   STATUS[84].EXT.Operation := FALSE;
   STATUS[84].EXT.Forced := TRUE;
   STATUS[84].EXT.BIT29 := FALSE;
   STATUS[84].EXT.BIT30 := FALSE;
   STATUS[84].EXT.BIT31 := FALSE;
   STATUS[84].EXT.ModeBit1 := FALSE;
   STATUS[84].EXT.ModeBit2 := FALSE;
   STATUS[84].EXT.ModeBit3 := FALSE;
   STATUS[84].EXT.BIT19 := FALSE;
   STATUS[84].EXT.BIT20 := FALSE;
   STATUS[84].EXT.AlarmSuppressed := FALSE;
   STATUS[84].EXT.AlarmPresent := FALSE;
   STATUS[84].EXT.AlarmFailUnAck := TRUE;
   STATUS[84].Status := 190;
   STATUS[84].TimeStamp := 16#1AEC;
   STATUS[85].EXT.AlarmWarnUnAck := FALSE;
   STATUS[85].EXT.AckRequired := FALSE;
   STATUS[85].EXT.Maintanence := FALSE;
   STATUS[85].EXT.Operation := TRUE;
   STATUS[85].EXT.Forced := FALSE;
   STATUS[85].EXT.BIT29 := FALSE;
   STATUS[85].EXT.BIT30 := FALSE;
   STATUS[85].EXT.BIT31 := FALSE;
   STATUS[85].EXT.ModeBit1 := FALSE;
   STATUS[85].EXT.ModeBit2 := FALSE;
   STATUS[85].EXT.ModeBit3 := FALSE;
   STATUS[85].EXT.BIT19 := FALSE;
   STATUS[85].EXT.BIT20 := FALSE;
   STATUS[85].EXT.AlarmSuppressed := FALSE;
   STATUS[85].EXT.AlarmPresent := FALSE;
   STATUS[85].EXT.AlarmFailUnAck := FALSE;
   STATUS[85].Status := 1;
   STATUS[85].TimeStamp := 16#3928;
   STATUS[86].EXT.AlarmWarnUnAck := FALSE;
   STATUS[86].EXT.AckRequired := FALSE;
   STATUS[86].EXT.Maintanence := FALSE;
   STATUS[86].EXT.Operation := TRUE;
   STATUS[86].EXT.Forced := FALSE;
   STATUS[86].EXT.BIT29 := FALSE;
   STATUS[86].EXT.BIT30 := FALSE;
   STATUS[86].EXT.BIT31 := FALSE;
   STATUS[86].EXT.ModeBit1 := FALSE;
   STATUS[86].EXT.ModeBit2 := FALSE;
   STATUS[86].EXT.ModeBit3 := FALSE;
   STATUS[86].EXT.BIT19 := FALSE;
   STATUS[86].EXT.BIT20 := FALSE;
   STATUS[86].EXT.AlarmSuppressed := FALSE;
   STATUS[86].EXT.AlarmPresent := FALSE;
   STATUS[86].EXT.AlarmFailUnAck := FALSE;
   STATUS[86].Status := 1;
   STATUS[86].TimeStamp := 16#3928;
   STATUS[87].EXT.AlarmWarnUnAck := FALSE;
   STATUS[87].EXT.AckRequired := FALSE;
   STATUS[87].EXT.Maintanence := FALSE;
   STATUS[87].EXT.Operation := FALSE;
   STATUS[87].EXT.Forced := FALSE;
   STATUS[87].EXT.BIT29 := FALSE;
   STATUS[87].EXT.BIT30 := FALSE;
   STATUS[87].EXT.BIT31 := FALSE;
   STATUS[87].EXT.ModeBit1 := FALSE;
   STATUS[87].EXT.ModeBit2 := FALSE;
   STATUS[87].EXT.ModeBit3 := FALSE;
   STATUS[87].EXT.BIT19 := FALSE;
   STATUS[87].EXT.BIT20 := FALSE;
   STATUS[87].EXT.AlarmSuppressed := TRUE;
   STATUS[87].EXT.AlarmPresent := FALSE;
   STATUS[87].EXT.AlarmFailUnAck := FALSE;
   STATUS[87].Status := 1;
   STATUS[87].TimeStamp := 16#84C0;
   STATUS[88].EXT.AlarmWarnUnAck := FALSE;
   STATUS[88].EXT.AckRequired := FALSE;
   STATUS[88].EXT.Maintanence := FALSE;
   STATUS[88].EXT.Operation := FALSE;
   STATUS[88].EXT.Forced := FALSE;
   STATUS[88].EXT.BIT29 := FALSE;
   STATUS[88].EXT.BIT30 := FALSE;
   STATUS[88].EXT.BIT31 := FALSE;
   STATUS[88].EXT.ModeBit1 := FALSE;
   STATUS[88].EXT.ModeBit2 := FALSE;
   STATUS[88].EXT.ModeBit3 := FALSE;
   STATUS[88].EXT.BIT19 := FALSE;
   STATUS[88].EXT.BIT20 := FALSE;
   STATUS[88].EXT.AlarmSuppressed := TRUE;
   STATUS[88].EXT.AlarmPresent := FALSE;
   STATUS[88].EXT.AlarmFailUnAck := FALSE;
   STATUS[88].Status := 1;
   STATUS[88].TimeStamp := 16#84BF;
   STATUS[89].EXT.AlarmWarnUnAck := FALSE;
   STATUS[89].EXT.AckRequired := FALSE;
   STATUS[89].EXT.Maintanence := FALSE;
   STATUS[89].EXT.Operation := FALSE;
   STATUS[89].EXT.Forced := TRUE;
   STATUS[89].EXT.BIT29 := FALSE;
   STATUS[89].EXT.BIT30 := FALSE;
   STATUS[89].EXT.BIT31 := FALSE;
   STATUS[89].EXT.ModeBit1 := FALSE;
   STATUS[89].EXT.ModeBit2 := FALSE;
   STATUS[89].EXT.ModeBit3 := FALSE;
   STATUS[89].EXT.BIT19 := FALSE;
   STATUS[89].EXT.BIT20 := FALSE;
   STATUS[89].EXT.AlarmSuppressed := FALSE;
   STATUS[89].EXT.AlarmPresent := FALSE;
   STATUS[89].EXT.AlarmFailUnAck := TRUE;
   STATUS[89].Status := 190;
   STATUS[89].TimeStamp := 16#71E9;
   STATUS[90].EXT.AlarmWarnUnAck := FALSE;
   STATUS[90].EXT.AckRequired := FALSE;
   STATUS[90].EXT.Maintanence := FALSE;
   STATUS[90].EXT.Operation := FALSE;
   STATUS[90].EXT.Forced := TRUE;
   STATUS[90].EXT.BIT29 := FALSE;
   STATUS[90].EXT.BIT30 := FALSE;
   STATUS[90].EXT.BIT31 := FALSE;
   STATUS[90].EXT.ModeBit1 := FALSE;
   STATUS[90].EXT.ModeBit2 := FALSE;
   STATUS[90].EXT.ModeBit3 := FALSE;
   STATUS[90].EXT.BIT19 := FALSE;
   STATUS[90].EXT.BIT20 := FALSE;
   STATUS[90].EXT.AlarmSuppressed := FALSE;
   STATUS[90].EXT.AlarmPresent := FALSE;
   STATUS[90].EXT.AlarmFailUnAck := TRUE;
   STATUS[90].Status := 190;
   STATUS[90].TimeStamp := 16#7C0C;
   STATUS[91].EXT.AlarmWarnUnAck := FALSE;
   STATUS[91].EXT.AckRequired := FALSE;
   STATUS[91].EXT.Maintanence := FALSE;
   STATUS[91].EXT.Operation := FALSE;
   STATUS[91].EXT.Forced := TRUE;
   STATUS[91].EXT.BIT29 := FALSE;
   STATUS[91].EXT.BIT30 := FALSE;
   STATUS[91].EXT.BIT31 := FALSE;
   STATUS[91].EXT.ModeBit1 := FALSE;
   STATUS[91].EXT.ModeBit2 := FALSE;
   STATUS[91].EXT.ModeBit3 := FALSE;
   STATUS[91].EXT.BIT19 := FALSE;
   STATUS[91].EXT.BIT20 := FALSE;
   STATUS[91].EXT.AlarmSuppressed := FALSE;
   STATUS[91].EXT.AlarmPresent := FALSE;
   STATUS[91].EXT.AlarmFailUnAck := TRUE;
   STATUS[91].Status := 190;
   STATUS[91].TimeStamp := 16#7882;
   STATUS[92].EXT.AlarmWarnUnAck := FALSE;
   STATUS[92].EXT.AckRequired := FALSE;
   STATUS[92].EXT.Maintanence := FALSE;
   STATUS[92].EXT.Operation := FALSE;
   STATUS[92].EXT.Forced := TRUE;
   STATUS[92].EXT.BIT29 := FALSE;
   STATUS[92].EXT.BIT30 := FALSE;
   STATUS[92].EXT.BIT31 := FALSE;
   STATUS[92].EXT.ModeBit1 := FALSE;
   STATUS[92].EXT.ModeBit2 := FALSE;
   STATUS[92].EXT.ModeBit3 := FALSE;
   STATUS[92].EXT.BIT19 := FALSE;
   STATUS[92].EXT.BIT20 := FALSE;
   STATUS[92].EXT.AlarmSuppressed := FALSE;
   STATUS[92].EXT.AlarmPresent := FALSE;
   STATUS[92].EXT.AlarmFailUnAck := TRUE;
   STATUS[92].Status := 190;
   STATUS[92].TimeStamp := 16#7534;
   STATUS[93].EXT.AlarmWarnUnAck := FALSE;
   STATUS[93].EXT.AckRequired := FALSE;
   STATUS[93].EXT.Maintanence := FALSE;
   STATUS[93].EXT.Operation := FALSE;
   STATUS[93].EXT.Forced := TRUE;
   STATUS[93].EXT.BIT29 := FALSE;
   STATUS[93].EXT.BIT30 := FALSE;
   STATUS[93].EXT.BIT31 := FALSE;
   STATUS[93].EXT.ModeBit1 := FALSE;
   STATUS[93].EXT.ModeBit2 := FALSE;
   STATUS[93].EXT.ModeBit3 := FALSE;
   STATUS[93].EXT.BIT19 := FALSE;
   STATUS[93].EXT.BIT20 := FALSE;
   STATUS[93].EXT.AlarmSuppressed := FALSE;
   STATUS[93].EXT.AlarmPresent := FALSE;
   STATUS[93].EXT.AlarmFailUnAck := TRUE;
   STATUS[93].Status := 190;
   STATUS[93].TimeStamp := 16#8187;
   STATUS[94].EXT.AlarmWarnUnAck := FALSE;
   STATUS[94].EXT.AckRequired := TRUE;
   STATUS[94].EXT.Maintanence := FALSE;
   STATUS[94].EXT.Operation := FALSE;
   STATUS[94].EXT.Forced := FALSE;
   STATUS[94].EXT.BIT29 := FALSE;
   STATUS[94].EXT.BIT30 := FALSE;
   STATUS[94].EXT.BIT31 := FALSE;
   STATUS[94].EXT.ModeBit1 := FALSE;
   STATUS[94].EXT.ModeBit2 := FALSE;
   STATUS[94].EXT.ModeBit3 := FALSE;
   STATUS[94].EXT.BIT19 := FALSE;
   STATUS[94].EXT.BIT20 := FALSE;
   STATUS[94].EXT.AlarmSuppressed := FALSE;
   STATUS[94].EXT.AlarmPresent := FALSE;
   STATUS[94].EXT.AlarmFailUnAck := TRUE;
   STATUS[94].Status := 231;
   STATUS[94].TimeStamp := 16#8854;
   STATUS[95].EXT.AlarmWarnUnAck := FALSE;
   STATUS[95].EXT.AckRequired := FALSE;
   STATUS[95].EXT.Maintanence := FALSE;
   STATUS[95].EXT.Operation := FALSE;
   STATUS[95].EXT.Forced := TRUE;
   STATUS[95].EXT.BIT29 := FALSE;
   STATUS[95].EXT.BIT30 := FALSE;
   STATUS[95].EXT.BIT31 := FALSE;
   STATUS[95].EXT.ModeBit1 := FALSE;
   STATUS[95].EXT.ModeBit2 := FALSE;
   STATUS[95].EXT.ModeBit3 := FALSE;
   STATUS[95].EXT.BIT19 := FALSE;
   STATUS[95].EXT.BIT20 := FALSE;
   STATUS[95].EXT.AlarmSuppressed := FALSE;
   STATUS[95].EXT.AlarmPresent := FALSE;
   STATUS[95].EXT.AlarmFailUnAck := TRUE;
   STATUS[95].Status := 190;
   STATUS[95].TimeStamp := 16#611D;
   STATUS[96].EXT.AlarmWarnUnAck := FALSE;
   STATUS[96].EXT.AckRequired := FALSE;
   STATUS[96].EXT.Maintanence := FALSE;
   STATUS[96].EXT.Operation := FALSE;
   STATUS[96].EXT.Forced := TRUE;
   STATUS[96].EXT.BIT29 := FALSE;
   STATUS[96].EXT.BIT30 := FALSE;
   STATUS[96].EXT.BIT31 := FALSE;
   STATUS[96].EXT.ModeBit1 := FALSE;
   STATUS[96].EXT.ModeBit2 := FALSE;
   STATUS[96].EXT.ModeBit3 := FALSE;
   STATUS[96].EXT.BIT19 := FALSE;
   STATUS[96].EXT.BIT20 := FALSE;
   STATUS[96].EXT.AlarmSuppressed := FALSE;
   STATUS[96].EXT.AlarmPresent := FALSE;
   STATUS[96].EXT.AlarmFailUnAck := TRUE;
   STATUS[96].Status := 190;
   STATUS[96].TimeStamp := 16#692D;
   STATUS[97].EXT.AlarmWarnUnAck := FALSE;
   STATUS[97].EXT.AckRequired := FALSE;
   STATUS[97].EXT.Maintanence := FALSE;
   STATUS[97].EXT.Operation := FALSE;
   STATUS[97].EXT.Forced := TRUE;
   STATUS[97].EXT.BIT29 := FALSE;
   STATUS[97].EXT.BIT30 := FALSE;
   STATUS[97].EXT.BIT31 := FALSE;
   STATUS[97].EXT.ModeBit1 := FALSE;
   STATUS[97].EXT.ModeBit2 := FALSE;
   STATUS[97].EXT.ModeBit3 := FALSE;
   STATUS[97].EXT.BIT19 := FALSE;
   STATUS[97].EXT.BIT20 := FALSE;
   STATUS[97].EXT.AlarmSuppressed := FALSE;
   STATUS[97].EXT.AlarmPresent := FALSE;
   STATUS[97].EXT.AlarmFailUnAck := TRUE;
   STATUS[97].Status := 190;
   STATUS[97].TimeStamp := 16#661E;
   STATUS[98].EXT.AlarmWarnUnAck := FALSE;
   STATUS[98].EXT.AckRequired := FALSE;
   STATUS[98].EXT.Maintanence := FALSE;
   STATUS[98].EXT.Operation := FALSE;
   STATUS[98].EXT.Forced := TRUE;
   STATUS[98].EXT.BIT29 := FALSE;
   STATUS[98].EXT.BIT30 := FALSE;
   STATUS[98].EXT.BIT31 := FALSE;
   STATUS[98].EXT.ModeBit1 := FALSE;
   STATUS[98].EXT.ModeBit2 := FALSE;
   STATUS[98].EXT.ModeBit3 := FALSE;
   STATUS[98].EXT.BIT19 := FALSE;
   STATUS[98].EXT.BIT20 := FALSE;
   STATUS[98].EXT.AlarmSuppressed := FALSE;
   STATUS[98].EXT.AlarmPresent := FALSE;
   STATUS[98].EXT.AlarmFailUnAck := TRUE;
   STATUS[98].Status := 190;
   STATUS[98].TimeStamp := 16#6F16;
   STATUS[99].EXT.AlarmWarnUnAck := FALSE;
   STATUS[99].EXT.AckRequired := FALSE;
   STATUS[99].EXT.Maintanence := FALSE;
   STATUS[99].EXT.Operation := FALSE;
   STATUS[99].EXT.Forced := TRUE;
   STATUS[99].EXT.BIT29 := FALSE;
   STATUS[99].EXT.BIT30 := FALSE;
   STATUS[99].EXT.BIT31 := FALSE;
   STATUS[99].EXT.ModeBit1 := FALSE;
   STATUS[99].EXT.ModeBit2 := FALSE;
   STATUS[99].EXT.ModeBit3 := FALSE;
   STATUS[99].EXT.BIT19 := FALSE;
   STATUS[99].EXT.BIT20 := FALSE;
   STATUS[99].EXT.AlarmSuppressed := FALSE;
   STATUS[99].EXT.AlarmPresent := FALSE;
   STATUS[99].EXT.AlarmFailUnAck := TRUE;
   STATUS[99].Status := 190;
   STATUS[99].TimeStamp := 16#4FA7;
   STATUS[100].EXT.AlarmWarnUnAck := FALSE;
   STATUS[100].EXT.AckRequired := FALSE;
   STATUS[100].EXT.Maintanence := FALSE;
   STATUS[100].EXT.Operation := FALSE;
   STATUS[100].EXT.Forced := TRUE;
   STATUS[100].EXT.BIT29 := FALSE;
   STATUS[100].EXT.BIT30 := FALSE;
   STATUS[100].EXT.BIT31 := FALSE;
   STATUS[100].EXT.ModeBit1 := FALSE;
   STATUS[100].EXT.ModeBit2 := FALSE;
   STATUS[100].EXT.ModeBit3 := FALSE;
   STATUS[100].EXT.BIT19 := FALSE;
   STATUS[100].EXT.BIT20 := FALSE;
   STATUS[100].EXT.AlarmSuppressed := FALSE;
   STATUS[100].EXT.AlarmPresent := FALSE;
   STATUS[100].EXT.AlarmFailUnAck := TRUE;
   STATUS[100].Status := 190;
   STATUS[100].TimeStamp := 16#8403;
   STATUS[101].EXT.AlarmWarnUnAck := FALSE;
   STATUS[101].EXT.AckRequired := FALSE;
   STATUS[101].EXT.Maintanence := FALSE;
   STATUS[101].EXT.Operation := FALSE;
   STATUS[101].EXT.Forced := TRUE;
   STATUS[101].EXT.BIT29 := FALSE;
   STATUS[101].EXT.BIT30 := FALSE;
   STATUS[101].EXT.BIT31 := FALSE;
   STATUS[101].EXT.ModeBit1 := FALSE;
   STATUS[101].EXT.ModeBit2 := FALSE;
   STATUS[101].EXT.ModeBit3 := FALSE;
   STATUS[101].EXT.BIT19 := FALSE;
   STATUS[101].EXT.BIT20 := FALSE;
   STATUS[101].EXT.AlarmSuppressed := FALSE;
   STATUS[101].EXT.AlarmPresent := FALSE;
   STATUS[101].EXT.AlarmFailUnAck := TRUE;
   STATUS[101].Status := 190;
   STATUS[101].TimeStamp := 16#6C19;
   STATUS[102].EXT.AlarmWarnUnAck := FALSE;
   STATUS[102].EXT.AckRequired := FALSE;
   STATUS[102].EXT.Maintanence := FALSE;
   STATUS[102].EXT.Operation := FALSE;
   STATUS[102].EXT.Forced := TRUE;
   STATUS[102].EXT.BIT29 := FALSE;
   STATUS[102].EXT.BIT30 := FALSE;
   STATUS[102].EXT.BIT31 := FALSE;
   STATUS[102].EXT.ModeBit1 := FALSE;
   STATUS[102].EXT.ModeBit2 := FALSE;
   STATUS[102].EXT.ModeBit3 := FALSE;
   STATUS[102].EXT.BIT19 := FALSE;
   STATUS[102].EXT.BIT20 := FALSE;
   STATUS[102].EXT.AlarmSuppressed := FALSE;
   STATUS[102].EXT.AlarmPresent := FALSE;
   STATUS[102].EXT.AlarmFailUnAck := TRUE;
   STATUS[102].Status := 190;
   STATUS[102].TimeStamp := 16#7EB8;
   STATUS[103].EXT.AlarmWarnUnAck := FALSE;
   STATUS[103].EXT.AckRequired := FALSE;
   STATUS[103].EXT.Maintanence := FALSE;
   STATUS[103].EXT.Operation := TRUE;
   STATUS[103].EXT.Forced := FALSE;
   STATUS[103].EXT.BIT29 := FALSE;
   STATUS[103].EXT.BIT30 := FALSE;
   STATUS[103].EXT.BIT31 := FALSE;
   STATUS[103].EXT.ModeBit1 := FALSE;
   STATUS[103].EXT.ModeBit2 := FALSE;
   STATUS[103].EXT.ModeBit3 := FALSE;
   STATUS[103].EXT.BIT19 := FALSE;
   STATUS[103].EXT.BIT20 := FALSE;
   STATUS[103].EXT.AlarmSuppressed := FALSE;
   STATUS[103].EXT.AlarmPresent := FALSE;
   STATUS[103].EXT.AlarmFailUnAck := FALSE;
   STATUS[103].Status := 1;
   STATUS[103].TimeStamp := 16#3928;
   STATUS[104].EXT.AlarmWarnUnAck := FALSE;
   STATUS[104].EXT.AckRequired := FALSE;
   STATUS[104].EXT.Maintanence := FALSE;
   STATUS[104].EXT.Operation := TRUE;
   STATUS[104].EXT.Forced := FALSE;
   STATUS[104].EXT.BIT29 := FALSE;
   STATUS[104].EXT.BIT30 := FALSE;
   STATUS[104].EXT.BIT31 := FALSE;
   STATUS[104].EXT.ModeBit1 := FALSE;
   STATUS[104].EXT.ModeBit2 := FALSE;
   STATUS[104].EXT.ModeBit3 := FALSE;
   STATUS[104].EXT.BIT19 := FALSE;
   STATUS[104].EXT.BIT20 := FALSE;
   STATUS[104].EXT.AlarmSuppressed := FALSE;
   STATUS[104].EXT.AlarmPresent := FALSE;
   STATUS[104].EXT.AlarmFailUnAck := FALSE;
   STATUS[104].Status := 1;
   STATUS[104].TimeStamp := 16#3928;
   STATUS[105].EXT.AlarmWarnUnAck := FALSE;
   STATUS[105].EXT.AckRequired := FALSE;
   STATUS[105].EXT.Maintanence := FALSE;
   STATUS[105].EXT.Operation := TRUE;
   STATUS[105].EXT.Forced := FALSE;
   STATUS[105].EXT.BIT29 := FALSE;
   STATUS[105].EXT.BIT30 := FALSE;
   STATUS[105].EXT.BIT31 := FALSE;
   STATUS[105].EXT.ModeBit1 := FALSE;
   STATUS[105].EXT.ModeBit2 := FALSE;
   STATUS[105].EXT.ModeBit3 := FALSE;
   STATUS[105].EXT.BIT19 := FALSE;
   STATUS[105].EXT.BIT20 := FALSE;
   STATUS[105].EXT.AlarmSuppressed := FALSE;
   STATUS[105].EXT.AlarmPresent := FALSE;
   STATUS[105].EXT.AlarmFailUnAck := FALSE;
   STATUS[105].Status := 1;
   STATUS[105].TimeStamp := 16#3928;
   STATUS[106].EXT.AlarmWarnUnAck := FALSE;
   STATUS[106].EXT.AckRequired := FALSE;
   STATUS[106].EXT.Maintanence := FALSE;
   STATUS[106].EXT.Operation := TRUE;
   STATUS[106].EXT.Forced := FALSE;
   STATUS[106].EXT.BIT29 := FALSE;
   STATUS[106].EXT.BIT30 := FALSE;
   STATUS[106].EXT.BIT31 := FALSE;
   STATUS[106].EXT.ModeBit1 := FALSE;
   STATUS[106].EXT.ModeBit2 := FALSE;
   STATUS[106].EXT.ModeBit3 := FALSE;
   STATUS[106].EXT.BIT19 := FALSE;
   STATUS[106].EXT.BIT20 := FALSE;
   STATUS[106].EXT.AlarmSuppressed := FALSE;
   STATUS[106].EXT.AlarmPresent := FALSE;
   STATUS[106].EXT.AlarmFailUnAck := FALSE;
   STATUS[106].Status := 1;
   STATUS[106].TimeStamp := 16#3928;
   STATUS[107].EXT.AlarmWarnUnAck := FALSE;
   STATUS[107].EXT.AckRequired := FALSE;
   STATUS[107].EXT.Maintanence := FALSE;
   STATUS[107].EXT.Operation := TRUE;
   STATUS[107].EXT.Forced := FALSE;
   STATUS[107].EXT.BIT29 := FALSE;
   STATUS[107].EXT.BIT30 := FALSE;
   STATUS[107].EXT.BIT31 := FALSE;
   STATUS[107].EXT.ModeBit1 := FALSE;
   STATUS[107].EXT.ModeBit2 := FALSE;
   STATUS[107].EXT.ModeBit3 := FALSE;
   STATUS[107].EXT.BIT19 := FALSE;
   STATUS[107].EXT.BIT20 := FALSE;
   STATUS[107].EXT.AlarmSuppressed := FALSE;
   STATUS[107].EXT.AlarmPresent := FALSE;
   STATUS[107].EXT.AlarmFailUnAck := FALSE;
   STATUS[107].Status := 1;
   STATUS[107].TimeStamp := 16#3928;
   STATUS[108].EXT.AlarmWarnUnAck := FALSE;
   STATUS[108].EXT.AckRequired := FALSE;
   STATUS[108].EXT.Maintanence := FALSE;
   STATUS[108].EXT.Operation := FALSE;
   STATUS[108].EXT.Forced := FALSE;
   STATUS[108].EXT.BIT29 := FALSE;
   STATUS[108].EXT.BIT30 := FALSE;
   STATUS[108].EXT.BIT31 := FALSE;
   STATUS[108].EXT.ModeBit1 := FALSE;
   STATUS[108].EXT.ModeBit2 := FALSE;
   STATUS[108].EXT.ModeBit3 := FALSE;
   STATUS[108].EXT.BIT19 := FALSE;
   STATUS[108].EXT.BIT20 := FALSE;
   STATUS[108].EXT.AlarmSuppressed := TRUE;
   STATUS[108].EXT.AlarmPresent := TRUE;
   STATUS[108].EXT.AlarmFailUnAck := TRUE;
   STATUS[108].Status := 201;
   STATUS[108].TimeStamp := 16#CE77;
   STATUS[109].EXT.AlarmWarnUnAck := FALSE;
   STATUS[109].EXT.AckRequired := FALSE;
   STATUS[109].EXT.Maintanence := FALSE;
   STATUS[109].EXT.Operation := FALSE;
   STATUS[109].EXT.Forced := TRUE;
   STATUS[109].EXT.BIT29 := FALSE;
   STATUS[109].EXT.BIT30 := FALSE;
   STATUS[109].EXT.BIT31 := FALSE;
   STATUS[109].EXT.ModeBit1 := FALSE;
   STATUS[109].EXT.ModeBit2 := FALSE;
   STATUS[109].EXT.ModeBit3 := FALSE;
   STATUS[109].EXT.BIT19 := FALSE;
   STATUS[109].EXT.BIT20 := FALSE;
   STATUS[109].EXT.AlarmSuppressed := FALSE;
   STATUS[109].EXT.AlarmPresent := FALSE;
   STATUS[109].EXT.AlarmFailUnAck := TRUE;
   STATUS[109].Status := 190;
   STATUS[109].TimeStamp := 16#D712;
   STATUS[110].EXT.AlarmWarnUnAck := FALSE;
   STATUS[110].EXT.AckRequired := FALSE;
   STATUS[110].EXT.Maintanence := FALSE;
   STATUS[110].EXT.Operation := FALSE;
   STATUS[110].EXT.Forced := TRUE;
   STATUS[110].EXT.BIT29 := FALSE;
   STATUS[110].EXT.BIT30 := FALSE;
   STATUS[110].EXT.BIT31 := FALSE;
   STATUS[110].EXT.ModeBit1 := FALSE;
   STATUS[110].EXT.ModeBit2 := FALSE;
   STATUS[110].EXT.ModeBit3 := FALSE;
   STATUS[110].EXT.BIT19 := FALSE;
   STATUS[110].EXT.BIT20 := FALSE;
   STATUS[110].EXT.AlarmSuppressed := FALSE;
   STATUS[110].EXT.AlarmPresent := FALSE;
   STATUS[110].EXT.AlarmFailUnAck := TRUE;
   STATUS[110].Status := 190;
   STATUS[110].TimeStamp := 16#969A;
   STATUS[111].EXT.AlarmWarnUnAck := FALSE;
   STATUS[111].EXT.AckRequired := FALSE;
   STATUS[111].EXT.Maintanence := FALSE;
   STATUS[111].EXT.Operation := FALSE;
   STATUS[111].EXT.Forced := FALSE;
   STATUS[111].EXT.BIT29 := FALSE;
   STATUS[111].EXT.BIT30 := FALSE;
   STATUS[111].EXT.BIT31 := FALSE;
   STATUS[111].EXT.ModeBit1 := FALSE;
   STATUS[111].EXT.ModeBit2 := FALSE;
   STATUS[111].EXT.ModeBit3 := FALSE;
   STATUS[111].EXT.BIT19 := FALSE;
   STATUS[111].EXT.BIT20 := FALSE;
   STATUS[111].EXT.AlarmSuppressed := TRUE;
   STATUS[111].EXT.AlarmPresent := FALSE;
   STATUS[111].EXT.AlarmFailUnAck := FALSE;
   STATUS[111].Status := 1;
   STATUS[111].TimeStamp := 16#9BB5;
   STATUS[112].EXT.AlarmWarnUnAck := FALSE;
   STATUS[112].EXT.AckRequired := FALSE;
   STATUS[112].EXT.Maintanence := FALSE;
   STATUS[112].EXT.Operation := FALSE;
   STATUS[112].EXT.Forced := TRUE;
   STATUS[112].EXT.BIT29 := FALSE;
   STATUS[112].EXT.BIT30 := FALSE;
   STATUS[112].EXT.BIT31 := FALSE;
   STATUS[112].EXT.ModeBit1 := FALSE;
   STATUS[112].EXT.ModeBit2 := FALSE;
   STATUS[112].EXT.ModeBit3 := FALSE;
   STATUS[112].EXT.BIT19 := FALSE;
   STATUS[112].EXT.BIT20 := FALSE;
   STATUS[112].EXT.AlarmSuppressed := FALSE;
   STATUS[112].EXT.AlarmPresent := FALSE;
   STATUS[112].EXT.AlarmFailUnAck := TRUE;
   STATUS[112].Status := 190;
   STATUS[112].TimeStamp := 16#87AE;
   STATUS[113].EXT.AlarmWarnUnAck := FALSE;
   STATUS[113].EXT.AckRequired := FALSE;
   STATUS[113].EXT.Maintanence := FALSE;
   STATUS[113].EXT.Operation := FALSE;
   STATUS[113].EXT.Forced := FALSE;
   STATUS[113].EXT.BIT29 := FALSE;
   STATUS[113].EXT.BIT30 := FALSE;
   STATUS[113].EXT.BIT31 := FALSE;
   STATUS[113].EXT.ModeBit1 := FALSE;
   STATUS[113].EXT.ModeBit2 := FALSE;
   STATUS[113].EXT.ModeBit3 := FALSE;
   STATUS[113].EXT.BIT19 := FALSE;
   STATUS[113].EXT.BIT20 := FALSE;
   STATUS[113].EXT.AlarmSuppressed := FALSE;
   STATUS[113].EXT.AlarmPresent := FALSE;
   STATUS[113].EXT.AlarmFailUnAck := FALSE;
   STATUS[113].Status := -22466;
   STATUS[113].TimeStamp := 16#84BA;
   STATUS[114].EXT.AlarmWarnUnAck := FALSE;
   STATUS[114].EXT.AckRequired := FALSE;
   STATUS[114].EXT.Maintanence := FALSE;
   STATUS[114].EXT.Operation := TRUE;
   STATUS[114].EXT.Forced := FALSE;
   STATUS[114].EXT.BIT29 := FALSE;
   STATUS[114].EXT.BIT30 := FALSE;
   STATUS[114].EXT.BIT31 := FALSE;
   STATUS[114].EXT.ModeBit1 := FALSE;
   STATUS[114].EXT.ModeBit2 := FALSE;
   STATUS[114].EXT.ModeBit3 := FALSE;
   STATUS[114].EXT.BIT19 := FALSE;
   STATUS[114].EXT.BIT20 := FALSE;
   STATUS[114].EXT.AlarmSuppressed := FALSE;
   STATUS[114].EXT.AlarmPresent := FALSE;
   STATUS[114].EXT.AlarmFailUnAck := FALSE;
   STATUS[114].Status := 4177;
   STATUS[114].TimeStamp := 16#583C;
   STATUS[115].EXT.AlarmWarnUnAck := FALSE;
   STATUS[115].EXT.AckRequired := FALSE;
   STATUS[115].EXT.Maintanence := FALSE;
   STATUS[115].EXT.Operation := TRUE;
   STATUS[115].EXT.Forced := FALSE;
   STATUS[115].EXT.BIT29 := FALSE;
   STATUS[115].EXT.BIT30 := FALSE;
   STATUS[115].EXT.BIT31 := FALSE;
   STATUS[115].EXT.ModeBit1 := FALSE;
   STATUS[115].EXT.ModeBit2 := FALSE;
   STATUS[115].EXT.ModeBit3 := FALSE;
   STATUS[115].EXT.BIT19 := FALSE;
   STATUS[115].EXT.BIT20 := FALSE;
   STATUS[115].EXT.AlarmSuppressed := FALSE;
   STATUS[115].EXT.AlarmPresent := FALSE;
   STATUS[115].EXT.AlarmFailUnAck := FALSE;
   STATUS[115].Status := 4177;
   STATUS[115].TimeStamp := 16#5ACA;
   STATUS[116].EXT.AlarmWarnUnAck := FALSE;
   STATUS[116].EXT.AckRequired := FALSE;
   STATUS[116].EXT.Maintanence := FALSE;
   STATUS[116].EXT.Operation := FALSE;
   STATUS[116].EXT.Forced := FALSE;
   STATUS[116].EXT.BIT29 := FALSE;
   STATUS[116].EXT.BIT30 := FALSE;
   STATUS[116].EXT.BIT31 := FALSE;
   STATUS[116].EXT.ModeBit1 := FALSE;
   STATUS[116].EXT.ModeBit2 := FALSE;
   STATUS[116].EXT.ModeBit3 := FALSE;
   STATUS[116].EXT.BIT19 := FALSE;
   STATUS[116].EXT.BIT20 := FALSE;
   STATUS[116].EXT.AlarmSuppressed := TRUE;
   STATUS[116].EXT.AlarmPresent := FALSE;
   STATUS[116].EXT.AlarmFailUnAck := FALSE;
   STATUS[116].Status := 1;
   STATUS[116].TimeStamp := 16#84BF;
   STATUS[117].EXT.AlarmWarnUnAck := FALSE;
   STATUS[117].EXT.AckRequired := FALSE;
   STATUS[117].EXT.Maintanence := FALSE;
   STATUS[117].EXT.Operation := FALSE;
   STATUS[117].EXT.Forced := FALSE;
   STATUS[117].EXT.BIT29 := FALSE;
   STATUS[117].EXT.BIT30 := FALSE;
   STATUS[117].EXT.BIT31 := FALSE;
   STATUS[117].EXT.ModeBit1 := FALSE;
   STATUS[117].EXT.ModeBit2 := FALSE;
   STATUS[117].EXT.ModeBit3 := FALSE;
   STATUS[117].EXT.BIT19 := FALSE;
   STATUS[117].EXT.BIT20 := FALSE;
   STATUS[117].EXT.AlarmSuppressed := TRUE;
   STATUS[117].EXT.AlarmPresent := TRUE;
   STATUS[117].EXT.AlarmFailUnAck := TRUE;
   STATUS[117].Status := 201;
   STATUS[117].TimeStamp := 16#E23A;
   STATUS[118].EXT.AlarmWarnUnAck := FALSE;
   STATUS[118].EXT.AckRequired := FALSE;
   STATUS[118].EXT.Maintanence := FALSE;
   STATUS[118].EXT.Operation := FALSE;
   STATUS[118].EXT.Forced := FALSE;
   STATUS[118].EXT.BIT29 := FALSE;
   STATUS[118].EXT.BIT30 := FALSE;
   STATUS[118].EXT.BIT31 := FALSE;
   STATUS[118].EXT.ModeBit1 := FALSE;
   STATUS[118].EXT.ModeBit2 := FALSE;
   STATUS[118].EXT.ModeBit3 := FALSE;
   STATUS[118].EXT.BIT19 := FALSE;
   STATUS[118].EXT.BIT20 := FALSE;
   STATUS[118].EXT.AlarmSuppressed := TRUE;
   STATUS[118].EXT.AlarmPresent := TRUE;
   STATUS[118].EXT.AlarmFailUnAck := TRUE;
   STATUS[118].Status := 212;
   STATUS[118].TimeStamp := 16#3928;
   STATUS[119].EXT.AlarmWarnUnAck := FALSE;
   STATUS[119].EXT.AckRequired := FALSE;
   STATUS[119].EXT.Maintanence := FALSE;
   STATUS[119].EXT.Operation := FALSE;
   STATUS[119].EXT.Forced := FALSE;
   STATUS[119].EXT.BIT29 := FALSE;
   STATUS[119].EXT.BIT30 := FALSE;
   STATUS[119].EXT.BIT31 := FALSE;
   STATUS[119].EXT.ModeBit1 := FALSE;
   STATUS[119].EXT.ModeBit2 := FALSE;
   STATUS[119].EXT.ModeBit3 := FALSE;
   STATUS[119].EXT.BIT19 := FALSE;
   STATUS[119].EXT.BIT20 := FALSE;
   STATUS[119].EXT.AlarmSuppressed := TRUE;
   STATUS[119].EXT.AlarmPresent := TRUE;
   STATUS[119].EXT.AlarmFailUnAck := TRUE;
   STATUS[119].Status := 212;
   STATUS[119].TimeStamp := 16#3928;
   STATUS[120].EXT.AlarmWarnUnAck := FALSE;
   STATUS[120].EXT.AckRequired := FALSE;
   STATUS[120].EXT.Maintanence := FALSE;
   STATUS[120].EXT.Operation := FALSE;
   STATUS[120].EXT.Forced := FALSE;
   STATUS[120].EXT.BIT29 := FALSE;
   STATUS[120].EXT.BIT30 := FALSE;
   STATUS[120].EXT.BIT31 := FALSE;
   STATUS[120].EXT.ModeBit1 := FALSE;
   STATUS[120].EXT.ModeBit2 := FALSE;
   STATUS[120].EXT.ModeBit3 := FALSE;
   STATUS[120].EXT.BIT19 := FALSE;
   STATUS[120].EXT.BIT20 := FALSE;
   STATUS[120].EXT.AlarmSuppressed := TRUE;
   STATUS[120].EXT.AlarmPresent := TRUE;
   STATUS[120].EXT.AlarmFailUnAck := TRUE;
   STATUS[120].Status := 212;
   STATUS[120].TimeStamp := 16#3928;
   STATUS[121].EXT.AlarmWarnUnAck := FALSE;
   STATUS[121].EXT.AckRequired := FALSE;
   STATUS[121].EXT.Maintanence := FALSE;
   STATUS[121].EXT.Operation := FALSE;
   STATUS[121].EXT.Forced := FALSE;
   STATUS[121].EXT.BIT29 := FALSE;
   STATUS[121].EXT.BIT30 := FALSE;
   STATUS[121].EXT.BIT31 := FALSE;
   STATUS[121].EXT.ModeBit1 := FALSE;
   STATUS[121].EXT.ModeBit2 := FALSE;
   STATUS[121].EXT.ModeBit3 := FALSE;
   STATUS[121].EXT.BIT19 := FALSE;
   STATUS[121].EXT.BIT20 := FALSE;
   STATUS[121].EXT.AlarmSuppressed := TRUE;
   STATUS[121].EXT.AlarmPresent := TRUE;
   STATUS[121].EXT.AlarmFailUnAck := TRUE;
   STATUS[121].Status := 212;
   STATUS[121].TimeStamp := 16#3928;
   STATUS[122].EXT.AlarmWarnUnAck := FALSE;
   STATUS[122].EXT.AckRequired := FALSE;
   STATUS[122].EXT.Maintanence := FALSE;
   STATUS[122].EXT.Operation := FALSE;
   STATUS[122].EXT.Forced := FALSE;
   STATUS[122].EXT.BIT29 := FALSE;
   STATUS[122].EXT.BIT30 := FALSE;
   STATUS[122].EXT.BIT31 := FALSE;
   STATUS[122].EXT.ModeBit1 := FALSE;
   STATUS[122].EXT.ModeBit2 := FALSE;
   STATUS[122].EXT.ModeBit3 := FALSE;
   STATUS[122].EXT.BIT19 := FALSE;
   STATUS[122].EXT.BIT20 := FALSE;
   STATUS[122].EXT.AlarmSuppressed := TRUE;
   STATUS[122].EXT.AlarmPresent := TRUE;
   STATUS[122].EXT.AlarmFailUnAck := TRUE;
   STATUS[122].Status := 212;
   STATUS[122].TimeStamp := 16#3928;
   STATUS[123].EXT.AlarmWarnUnAck := FALSE;
   STATUS[123].EXT.AckRequired := FALSE;
   STATUS[123].EXT.Maintanence := FALSE;
   STATUS[123].EXT.Operation := FALSE;
   STATUS[123].EXT.Forced := FALSE;
   STATUS[123].EXT.BIT29 := FALSE;
   STATUS[123].EXT.BIT30 := FALSE;
   STATUS[123].EXT.BIT31 := FALSE;
   STATUS[123].EXT.ModeBit1 := FALSE;
   STATUS[123].EXT.ModeBit2 := FALSE;
   STATUS[123].EXT.ModeBit3 := FALSE;
   STATUS[123].EXT.BIT19 := FALSE;
   STATUS[123].EXT.BIT20 := FALSE;
   STATUS[123].EXT.AlarmSuppressed := TRUE;
   STATUS[123].EXT.AlarmPresent := TRUE;
   STATUS[123].EXT.AlarmFailUnAck := TRUE;
   STATUS[123].Status := 207;
   STATUS[123].TimeStamp := 16#84C0;
   STATUS[124].EXT.AlarmWarnUnAck := FALSE;
   STATUS[124].EXT.AckRequired := FALSE;
   STATUS[124].EXT.Maintanence := FALSE;
   STATUS[124].EXT.Operation := TRUE;
   STATUS[124].EXT.Forced := FALSE;
   STATUS[124].EXT.BIT29 := FALSE;
   STATUS[124].EXT.BIT30 := FALSE;
   STATUS[124].EXT.BIT31 := FALSE;
   STATUS[124].EXT.ModeBit1 := FALSE;
   STATUS[124].EXT.ModeBit2 := FALSE;
   STATUS[124].EXT.ModeBit3 := FALSE;
   STATUS[124].EXT.BIT19 := FALSE;
   STATUS[124].EXT.BIT20 := FALSE;
   STATUS[124].EXT.AlarmSuppressed := FALSE;
   STATUS[124].EXT.AlarmPresent := FALSE;
   STATUS[124].EXT.AlarmFailUnAck := FALSE;
   STATUS[124].Status := 1;
   STATUS[124].TimeStamp := 16#3928;
   STATUS[125].EXT.AlarmWarnUnAck := FALSE;
   STATUS[125].EXT.AckRequired := FALSE;
   STATUS[125].EXT.Maintanence := FALSE;
   STATUS[125].EXT.Operation := FALSE;
   STATUS[125].EXT.Forced := FALSE;
   STATUS[125].EXT.BIT29 := FALSE;
   STATUS[125].EXT.BIT30 := FALSE;
   STATUS[125].EXT.BIT31 := FALSE;
   STATUS[125].EXT.ModeBit1 := FALSE;
   STATUS[125].EXT.ModeBit2 := FALSE;
   STATUS[125].EXT.ModeBit3 := FALSE;
   STATUS[125].EXT.BIT19 := FALSE;
   STATUS[125].EXT.BIT20 := FALSE;
   STATUS[125].EXT.AlarmSuppressed := FALSE;
   STATUS[125].EXT.AlarmPresent := FALSE;
   STATUS[125].EXT.AlarmFailUnAck := FALSE;
   STATUS[125].Status := 0;
   STATUS[125].TimeStamp := 16#0000;
   STATUS[126].EXT.AlarmWarnUnAck := FALSE;
   STATUS[126].EXT.AckRequired := FALSE;
   STATUS[126].EXT.Maintanence := FALSE;
   STATUS[126].EXT.Operation := FALSE;
   STATUS[126].EXT.Forced := FALSE;
   STATUS[126].EXT.BIT29 := FALSE;
   STATUS[126].EXT.BIT30 := FALSE;
   STATUS[126].EXT.BIT31 := FALSE;
   STATUS[126].EXT.ModeBit1 := FALSE;
   STATUS[126].EXT.ModeBit2 := FALSE;
   STATUS[126].EXT.ModeBit3 := FALSE;
   STATUS[126].EXT.BIT19 := FALSE;
   STATUS[126].EXT.BIT20 := FALSE;
   STATUS[126].EXT.AlarmSuppressed := FALSE;
   STATUS[126].EXT.AlarmPresent := FALSE;
   STATUS[126].EXT.AlarmFailUnAck := FALSE;
   STATUS[126].Status := 0;
   STATUS[126].TimeStamp := 16#0000;
   STATUS[127].EXT.AlarmWarnUnAck := FALSE;
   STATUS[127].EXT.AckRequired := FALSE;
   STATUS[127].EXT.Maintanence := FALSE;
   STATUS[127].EXT.Operation := FALSE;
   STATUS[127].EXT.Forced := FALSE;
   STATUS[127].EXT.BIT29 := FALSE;
   STATUS[127].EXT.BIT30 := FALSE;
   STATUS[127].EXT.BIT31 := FALSE;
   STATUS[127].EXT.ModeBit1 := FALSE;
   STATUS[127].EXT.ModeBit2 := FALSE;
   STATUS[127].EXT.ModeBit3 := FALSE;
   STATUS[127].EXT.BIT19 := FALSE;
   STATUS[127].EXT.BIT20 := FALSE;
   STATUS[127].EXT.AlarmSuppressed := FALSE;
   STATUS[127].EXT.AlarmPresent := FALSE;
   STATUS[127].EXT.AlarmFailUnAck := FALSE;
   STATUS[127].Status := 0;
   STATUS[127].TimeStamp := 16#0000;
   STATUS[128].EXT.AlarmWarnUnAck := FALSE;
   STATUS[128].EXT.AckRequired := FALSE;
   STATUS[128].EXT.Maintanence := FALSE;
   STATUS[128].EXT.Operation := FALSE;
   STATUS[128].EXT.Forced := FALSE;
   STATUS[128].EXT.BIT29 := FALSE;
   STATUS[128].EXT.BIT30 := FALSE;
   STATUS[128].EXT.BIT31 := FALSE;
   STATUS[128].EXT.ModeBit1 := FALSE;
   STATUS[128].EXT.ModeBit2 := FALSE;
   STATUS[128].EXT.ModeBit3 := FALSE;
   STATUS[128].EXT.BIT19 := FALSE;
   STATUS[128].EXT.BIT20 := FALSE;
   STATUS[128].EXT.AlarmSuppressed := FALSE;
   STATUS[128].EXT.AlarmPresent := FALSE;
   STATUS[128].EXT.AlarmFailUnAck := FALSE;
   STATUS[128].Status := 0;
   STATUS[128].TimeStamp := 16#0000;
   STATUS[129].EXT.AlarmWarnUnAck := FALSE;
   STATUS[129].EXT.AckRequired := FALSE;
   STATUS[129].EXT.Maintanence := FALSE;
   STATUS[129].EXT.Operation := FALSE;
   STATUS[129].EXT.Forced := FALSE;
   STATUS[129].EXT.BIT29 := FALSE;
   STATUS[129].EXT.BIT30 := FALSE;
   STATUS[129].EXT.BIT31 := FALSE;
   STATUS[129].EXT.ModeBit1 := FALSE;
   STATUS[129].EXT.ModeBit2 := FALSE;
   STATUS[129].EXT.ModeBit3 := FALSE;
   STATUS[129].EXT.BIT19 := FALSE;
   STATUS[129].EXT.BIT20 := FALSE;
   STATUS[129].EXT.AlarmSuppressed := FALSE;
   STATUS[129].EXT.AlarmPresent := FALSE;
   STATUS[129].EXT.AlarmFailUnAck := FALSE;
   STATUS[129].Status := 0;
   STATUS[129].TimeStamp := 16#0000;
   STATUS[130].EXT.AlarmWarnUnAck := FALSE;
   STATUS[130].EXT.AckRequired := FALSE;
   STATUS[130].EXT.Maintanence := FALSE;
   STATUS[130].EXT.Operation := FALSE;
   STATUS[130].EXT.Forced := FALSE;
   STATUS[130].EXT.BIT29 := FALSE;
   STATUS[130].EXT.BIT30 := FALSE;
   STATUS[130].EXT.BIT31 := FALSE;
   STATUS[130].EXT.ModeBit1 := FALSE;
   STATUS[130].EXT.ModeBit2 := FALSE;
   STATUS[130].EXT.ModeBit3 := FALSE;
   STATUS[130].EXT.BIT19 := FALSE;
   STATUS[130].EXT.BIT20 := FALSE;
   STATUS[130].EXT.AlarmSuppressed := FALSE;
   STATUS[130].EXT.AlarmPresent := FALSE;
   STATUS[130].EXT.AlarmFailUnAck := FALSE;
   STATUS[130].Status := 0;
   STATUS[130].TimeStamp := 16#0000;
   STATUS[131].EXT.AlarmWarnUnAck := FALSE;
   STATUS[131].EXT.AckRequired := FALSE;
   STATUS[131].EXT.Maintanence := FALSE;
   STATUS[131].EXT.Operation := FALSE;
   STATUS[131].EXT.Forced := FALSE;
   STATUS[131].EXT.BIT29 := FALSE;
   STATUS[131].EXT.BIT30 := FALSE;
   STATUS[131].EXT.BIT31 := FALSE;
   STATUS[131].EXT.ModeBit1 := FALSE;
   STATUS[131].EXT.ModeBit2 := FALSE;
   STATUS[131].EXT.ModeBit3 := FALSE;
   STATUS[131].EXT.BIT19 := FALSE;
   STATUS[131].EXT.BIT20 := FALSE;
   STATUS[131].EXT.AlarmSuppressed := FALSE;
   STATUS[131].EXT.AlarmPresent := FALSE;
   STATUS[131].EXT.AlarmFailUnAck := FALSE;
   STATUS[131].Status := 0;
   STATUS[131].TimeStamp := 16#0000;
   STATUS[132].EXT.AlarmWarnUnAck := FALSE;
   STATUS[132].EXT.AckRequired := FALSE;
   STATUS[132].EXT.Maintanence := FALSE;
   STATUS[132].EXT.Operation := FALSE;
   STATUS[132].EXT.Forced := FALSE;
   STATUS[132].EXT.BIT29 := FALSE;
   STATUS[132].EXT.BIT30 := FALSE;
   STATUS[132].EXT.BIT31 := FALSE;
   STATUS[132].EXT.ModeBit1 := FALSE;
   STATUS[132].EXT.ModeBit2 := FALSE;
   STATUS[132].EXT.ModeBit3 := FALSE;
   STATUS[132].EXT.BIT19 := FALSE;
   STATUS[132].EXT.BIT20 := FALSE;
   STATUS[132].EXT.AlarmSuppressed := FALSE;
   STATUS[132].EXT.AlarmPresent := FALSE;
   STATUS[132].EXT.AlarmFailUnAck := FALSE;
   STATUS[132].Status := 0;
   STATUS[132].TimeStamp := 16#0000;
   STATUS[133].EXT.AlarmWarnUnAck := FALSE;
   STATUS[133].EXT.AckRequired := FALSE;
   STATUS[133].EXT.Maintanence := FALSE;
   STATUS[133].EXT.Operation := FALSE;
   STATUS[133].EXT.Forced := FALSE;
   STATUS[133].EXT.BIT29 := FALSE;
   STATUS[133].EXT.BIT30 := FALSE;
   STATUS[133].EXT.BIT31 := FALSE;
   STATUS[133].EXT.ModeBit1 := FALSE;
   STATUS[133].EXT.ModeBit2 := FALSE;
   STATUS[133].EXT.ModeBit3 := FALSE;
   STATUS[133].EXT.BIT19 := FALSE;
   STATUS[133].EXT.BIT20 := FALSE;
   STATUS[133].EXT.AlarmSuppressed := FALSE;
   STATUS[133].EXT.AlarmPresent := FALSE;
   STATUS[133].EXT.AlarmFailUnAck := FALSE;
   STATUS[133].Status := 0;
   STATUS[133].TimeStamp := 16#0000;
   STATUS[134].EXT.AlarmWarnUnAck := FALSE;
   STATUS[134].EXT.AckRequired := FALSE;
   STATUS[134].EXT.Maintanence := FALSE;
   STATUS[134].EXT.Operation := FALSE;
   STATUS[134].EXT.Forced := FALSE;
   STATUS[134].EXT.BIT29 := FALSE;
   STATUS[134].EXT.BIT30 := FALSE;
   STATUS[134].EXT.BIT31 := FALSE;
   STATUS[134].EXT.ModeBit1 := FALSE;
   STATUS[134].EXT.ModeBit2 := FALSE;
   STATUS[134].EXT.ModeBit3 := FALSE;
   STATUS[134].EXT.BIT19 := FALSE;
   STATUS[134].EXT.BIT20 := FALSE;
   STATUS[134].EXT.AlarmSuppressed := FALSE;
   STATUS[134].EXT.AlarmPresent := FALSE;
   STATUS[134].EXT.AlarmFailUnAck := FALSE;
   STATUS[134].Status := 0;
   STATUS[134].TimeStamp := 16#0000;
   STATUS[135].EXT.AlarmWarnUnAck := FALSE;
   STATUS[135].EXT.AckRequired := FALSE;
   STATUS[135].EXT.Maintanence := FALSE;
   STATUS[135].EXT.Operation := FALSE;
   STATUS[135].EXT.Forced := FALSE;
   STATUS[135].EXT.BIT29 := FALSE;
   STATUS[135].EXT.BIT30 := FALSE;
   STATUS[135].EXT.BIT31 := FALSE;
   STATUS[135].EXT.ModeBit1 := FALSE;
   STATUS[135].EXT.ModeBit2 := FALSE;
   STATUS[135].EXT.ModeBit3 := FALSE;
   STATUS[135].EXT.BIT19 := FALSE;
   STATUS[135].EXT.BIT20 := FALSE;
   STATUS[135].EXT.AlarmSuppressed := FALSE;
   STATUS[135].EXT.AlarmPresent := FALSE;
   STATUS[135].EXT.AlarmFailUnAck := FALSE;
   STATUS[135].Status := 0;
   STATUS[135].TimeStamp := 16#0000;
   STATUS[136].EXT.AlarmWarnUnAck := FALSE;
   STATUS[136].EXT.AckRequired := FALSE;
   STATUS[136].EXT.Maintanence := FALSE;
   STATUS[136].EXT.Operation := FALSE;
   STATUS[136].EXT.Forced := FALSE;
   STATUS[136].EXT.BIT29 := FALSE;
   STATUS[136].EXT.BIT30 := FALSE;
   STATUS[136].EXT.BIT31 := FALSE;
   STATUS[136].EXT.ModeBit1 := FALSE;
   STATUS[136].EXT.ModeBit2 := FALSE;
   STATUS[136].EXT.ModeBit3 := FALSE;
   STATUS[136].EXT.BIT19 := FALSE;
   STATUS[136].EXT.BIT20 := FALSE;
   STATUS[136].EXT.AlarmSuppressed := FALSE;
   STATUS[136].EXT.AlarmPresent := FALSE;
   STATUS[136].EXT.AlarmFailUnAck := FALSE;
   STATUS[136].Status := 0;
   STATUS[136].TimeStamp := 16#0000;
   STATUS[137].EXT.AlarmWarnUnAck := FALSE;
   STATUS[137].EXT.AckRequired := FALSE;
   STATUS[137].EXT.Maintanence := FALSE;
   STATUS[137].EXT.Operation := FALSE;
   STATUS[137].EXT.Forced := FALSE;
   STATUS[137].EXT.BIT29 := FALSE;
   STATUS[137].EXT.BIT30 := FALSE;
   STATUS[137].EXT.BIT31 := FALSE;
   STATUS[137].EXT.ModeBit1 := FALSE;
   STATUS[137].EXT.ModeBit2 := FALSE;
   STATUS[137].EXT.ModeBit3 := FALSE;
   STATUS[137].EXT.BIT19 := FALSE;
   STATUS[137].EXT.BIT20 := FALSE;
   STATUS[137].EXT.AlarmSuppressed := FALSE;
   STATUS[137].EXT.AlarmPresent := FALSE;
   STATUS[137].EXT.AlarmFailUnAck := FALSE;
   STATUS[137].Status := 0;
   STATUS[137].TimeStamp := 16#0000;
   STATUS[138].EXT.AlarmWarnUnAck := FALSE;
   STATUS[138].EXT.AckRequired := FALSE;
   STATUS[138].EXT.Maintanence := FALSE;
   STATUS[138].EXT.Operation := FALSE;
   STATUS[138].EXT.Forced := FALSE;
   STATUS[138].EXT.BIT29 := FALSE;
   STATUS[138].EXT.BIT30 := FALSE;
   STATUS[138].EXT.BIT31 := FALSE;
   STATUS[138].EXT.ModeBit1 := FALSE;
   STATUS[138].EXT.ModeBit2 := FALSE;
   STATUS[138].EXT.ModeBit3 := FALSE;
   STATUS[138].EXT.BIT19 := FALSE;
   STATUS[138].EXT.BIT20 := FALSE;
   STATUS[138].EXT.AlarmSuppressed := FALSE;
   STATUS[138].EXT.AlarmPresent := FALSE;
   STATUS[138].EXT.AlarmFailUnAck := FALSE;
   STATUS[138].Status := 0;
   STATUS[138].TimeStamp := 16#0000;
   STATUS[139].EXT.AlarmWarnUnAck := FALSE;
   STATUS[139].EXT.AckRequired := FALSE;
   STATUS[139].EXT.Maintanence := FALSE;
   STATUS[139].EXT.Operation := FALSE;
   STATUS[139].EXT.Forced := FALSE;
   STATUS[139].EXT.BIT29 := FALSE;
   STATUS[139].EXT.BIT30 := FALSE;
   STATUS[139].EXT.BIT31 := FALSE;
   STATUS[139].EXT.ModeBit1 := FALSE;
   STATUS[139].EXT.ModeBit2 := FALSE;
   STATUS[139].EXT.ModeBit3 := FALSE;
   STATUS[139].EXT.BIT19 := FALSE;
   STATUS[139].EXT.BIT20 := FALSE;
   STATUS[139].EXT.AlarmSuppressed := FALSE;
   STATUS[139].EXT.AlarmPresent := FALSE;
   STATUS[139].EXT.AlarmFailUnAck := FALSE;
   STATUS[139].Status := 0;
   STATUS[139].TimeStamp := 16#0000;
   STATUS[140].EXT.AlarmWarnUnAck := FALSE;
   STATUS[140].EXT.AckRequired := FALSE;
   STATUS[140].EXT.Maintanence := FALSE;
   STATUS[140].EXT.Operation := FALSE;
   STATUS[140].EXT.Forced := FALSE;
   STATUS[140].EXT.BIT29 := FALSE;
   STATUS[140].EXT.BIT30 := FALSE;
   STATUS[140].EXT.BIT31 := FALSE;
   STATUS[140].EXT.ModeBit1 := FALSE;
   STATUS[140].EXT.ModeBit2 := FALSE;
   STATUS[140].EXT.ModeBit3 := FALSE;
   STATUS[140].EXT.BIT19 := FALSE;
   STATUS[140].EXT.BIT20 := FALSE;
   STATUS[140].EXT.AlarmSuppressed := FALSE;
   STATUS[140].EXT.AlarmPresent := FALSE;
   STATUS[140].EXT.AlarmFailUnAck := FALSE;
   STATUS[140].Status := 0;
   STATUS[140].TimeStamp := 16#0000;
   STATUS[141].EXT.AlarmWarnUnAck := FALSE;
   STATUS[141].EXT.AckRequired := FALSE;
   STATUS[141].EXT.Maintanence := FALSE;
   STATUS[141].EXT.Operation := FALSE;
   STATUS[141].EXT.Forced := FALSE;
   STATUS[141].EXT.BIT29 := FALSE;
   STATUS[141].EXT.BIT30 := FALSE;
   STATUS[141].EXT.BIT31 := FALSE;
   STATUS[141].EXT.ModeBit1 := FALSE;
   STATUS[141].EXT.ModeBit2 := FALSE;
   STATUS[141].EXT.ModeBit3 := FALSE;
   STATUS[141].EXT.BIT19 := FALSE;
   STATUS[141].EXT.BIT20 := FALSE;
   STATUS[141].EXT.AlarmSuppressed := FALSE;
   STATUS[141].EXT.AlarmPresent := FALSE;
   STATUS[141].EXT.AlarmFailUnAck := FALSE;
   STATUS[141].Status := 0;
   STATUS[141].TimeStamp := 16#0000;
   STATUS[142].EXT.AlarmWarnUnAck := FALSE;
   STATUS[142].EXT.AckRequired := FALSE;
   STATUS[142].EXT.Maintanence := FALSE;
   STATUS[142].EXT.Operation := FALSE;
   STATUS[142].EXT.Forced := FALSE;
   STATUS[142].EXT.BIT29 := FALSE;
   STATUS[142].EXT.BIT30 := FALSE;
   STATUS[142].EXT.BIT31 := FALSE;
   STATUS[142].EXT.ModeBit1 := FALSE;
   STATUS[142].EXT.ModeBit2 := FALSE;
   STATUS[142].EXT.ModeBit3 := FALSE;
   STATUS[142].EXT.BIT19 := FALSE;
   STATUS[142].EXT.BIT20 := FALSE;
   STATUS[142].EXT.AlarmSuppressed := FALSE;
   STATUS[142].EXT.AlarmPresent := FALSE;
   STATUS[142].EXT.AlarmFailUnAck := FALSE;
   STATUS[142].Status := 0;
   STATUS[142].TimeStamp := 16#0000;
   STATUS[143].EXT.AlarmWarnUnAck := FALSE;
   STATUS[143].EXT.AckRequired := FALSE;
   STATUS[143].EXT.Maintanence := FALSE;
   STATUS[143].EXT.Operation := FALSE;
   STATUS[143].EXT.Forced := FALSE;
   STATUS[143].EXT.BIT29 := FALSE;
   STATUS[143].EXT.BIT30 := FALSE;
   STATUS[143].EXT.BIT31 := FALSE;
   STATUS[143].EXT.ModeBit1 := FALSE;
   STATUS[143].EXT.ModeBit2 := FALSE;
   STATUS[143].EXT.ModeBit3 := FALSE;
   STATUS[143].EXT.BIT19 := FALSE;
   STATUS[143].EXT.BIT20 := FALSE;
   STATUS[143].EXT.AlarmSuppressed := FALSE;
   STATUS[143].EXT.AlarmPresent := FALSE;
   STATUS[143].EXT.AlarmFailUnAck := FALSE;
   STATUS[143].Status := 0;
   STATUS[143].TimeStamp := 16#0000;
   STATUS[144].EXT.AlarmWarnUnAck := FALSE;
   STATUS[144].EXT.AckRequired := FALSE;
   STATUS[144].EXT.Maintanence := FALSE;
   STATUS[144].EXT.Operation := FALSE;
   STATUS[144].EXT.Forced := FALSE;
   STATUS[144].EXT.BIT29 := FALSE;
   STATUS[144].EXT.BIT30 := FALSE;
   STATUS[144].EXT.BIT31 := FALSE;
   STATUS[144].EXT.ModeBit1 := FALSE;
   STATUS[144].EXT.ModeBit2 := FALSE;
   STATUS[144].EXT.ModeBit3 := FALSE;
   STATUS[144].EXT.BIT19 := FALSE;
   STATUS[144].EXT.BIT20 := FALSE;
   STATUS[144].EXT.AlarmSuppressed := FALSE;
   STATUS[144].EXT.AlarmPresent := FALSE;
   STATUS[144].EXT.AlarmFailUnAck := FALSE;
   STATUS[144].Status := 0;
   STATUS[144].TimeStamp := 16#0000;
   STATUS[145].EXT.AlarmWarnUnAck := FALSE;
   STATUS[145].EXT.AckRequired := FALSE;
   STATUS[145].EXT.Maintanence := FALSE;
   STATUS[145].EXT.Operation := FALSE;
   STATUS[145].EXT.Forced := FALSE;
   STATUS[145].EXT.BIT29 := FALSE;
   STATUS[145].EXT.BIT30 := FALSE;
   STATUS[145].EXT.BIT31 := FALSE;
   STATUS[145].EXT.ModeBit1 := FALSE;
   STATUS[145].EXT.ModeBit2 := FALSE;
   STATUS[145].EXT.ModeBit3 := FALSE;
   STATUS[145].EXT.BIT19 := FALSE;
   STATUS[145].EXT.BIT20 := FALSE;
   STATUS[145].EXT.AlarmSuppressed := FALSE;
   STATUS[145].EXT.AlarmPresent := FALSE;
   STATUS[145].EXT.AlarmFailUnAck := FALSE;
   STATUS[145].Status := 0;
   STATUS[145].TimeStamp := 16#0000;
   STATUS[146].EXT.AlarmWarnUnAck := FALSE;
   STATUS[146].EXT.AckRequired := FALSE;
   STATUS[146].EXT.Maintanence := FALSE;
   STATUS[146].EXT.Operation := FALSE;
   STATUS[146].EXT.Forced := FALSE;
   STATUS[146].EXT.BIT29 := FALSE;
   STATUS[146].EXT.BIT30 := FALSE;
   STATUS[146].EXT.BIT31 := FALSE;
   STATUS[146].EXT.ModeBit1 := FALSE;
   STATUS[146].EXT.ModeBit2 := FALSE;
   STATUS[146].EXT.ModeBit3 := FALSE;
   STATUS[146].EXT.BIT19 := FALSE;
   STATUS[146].EXT.BIT20 := FALSE;
   STATUS[146].EXT.AlarmSuppressed := FALSE;
   STATUS[146].EXT.AlarmPresent := FALSE;
   STATUS[146].EXT.AlarmFailUnAck := FALSE;
   STATUS[146].Status := 0;
   STATUS[146].TimeStamp := 16#0000;
   STATUS[147].EXT.AlarmWarnUnAck := FALSE;
   STATUS[147].EXT.AckRequired := FALSE;
   STATUS[147].EXT.Maintanence := FALSE;
   STATUS[147].EXT.Operation := FALSE;
   STATUS[147].EXT.Forced := FALSE;
   STATUS[147].EXT.BIT29 := FALSE;
   STATUS[147].EXT.BIT30 := FALSE;
   STATUS[147].EXT.BIT31 := FALSE;
   STATUS[147].EXT.ModeBit1 := FALSE;
   STATUS[147].EXT.ModeBit2 := FALSE;
   STATUS[147].EXT.ModeBit3 := FALSE;
   STATUS[147].EXT.BIT19 := FALSE;
   STATUS[147].EXT.BIT20 := FALSE;
   STATUS[147].EXT.AlarmSuppressed := FALSE;
   STATUS[147].EXT.AlarmPresent := FALSE;
   STATUS[147].EXT.AlarmFailUnAck := FALSE;
   STATUS[147].Status := 0;
   STATUS[147].TimeStamp := 16#0000;
   STATUS[148].EXT.AlarmWarnUnAck := FALSE;
   STATUS[148].EXT.AckRequired := FALSE;
   STATUS[148].EXT.Maintanence := FALSE;
   STATUS[148].EXT.Operation := FALSE;
   STATUS[148].EXT.Forced := FALSE;
   STATUS[148].EXT.BIT29 := FALSE;
   STATUS[148].EXT.BIT30 := FALSE;
   STATUS[148].EXT.BIT31 := FALSE;
   STATUS[148].EXT.ModeBit1 := FALSE;
   STATUS[148].EXT.ModeBit2 := FALSE;
   STATUS[148].EXT.ModeBit3 := FALSE;
   STATUS[148].EXT.BIT19 := FALSE;
   STATUS[148].EXT.BIT20 := FALSE;
   STATUS[148].EXT.AlarmSuppressed := FALSE;
   STATUS[148].EXT.AlarmPresent := FALSE;
   STATUS[148].EXT.AlarmFailUnAck := FALSE;
   STATUS[148].Status := 0;
   STATUS[148].TimeStamp := 16#0000;
   STATUS[149].EXT.AlarmWarnUnAck := FALSE;
   STATUS[149].EXT.AckRequired := FALSE;
   STATUS[149].EXT.Maintanence := FALSE;
   STATUS[149].EXT.Operation := FALSE;
   STATUS[149].EXT.Forced := FALSE;
   STATUS[149].EXT.BIT29 := FALSE;
   STATUS[149].EXT.BIT30 := FALSE;
   STATUS[149].EXT.BIT31 := FALSE;
   STATUS[149].EXT.ModeBit1 := FALSE;
   STATUS[149].EXT.ModeBit2 := FALSE;
   STATUS[149].EXT.ModeBit3 := FALSE;
   STATUS[149].EXT.BIT19 := FALSE;
   STATUS[149].EXT.BIT20 := FALSE;
   STATUS[149].EXT.AlarmSuppressed := FALSE;
   STATUS[149].EXT.AlarmPresent := FALSE;
   STATUS[149].EXT.AlarmFailUnAck := FALSE;
   STATUS[149].Status := 0;
   STATUS[149].TimeStamp := 16#0000;
   STATUS[150].EXT.AlarmWarnUnAck := FALSE;
   STATUS[150].EXT.AckRequired := FALSE;
   STATUS[150].EXT.Maintanence := FALSE;
   STATUS[150].EXT.Operation := FALSE;
   STATUS[150].EXT.Forced := FALSE;
   STATUS[150].EXT.BIT29 := FALSE;
   STATUS[150].EXT.BIT30 := FALSE;
   STATUS[150].EXT.BIT31 := FALSE;
   STATUS[150].EXT.ModeBit1 := FALSE;
   STATUS[150].EXT.ModeBit2 := FALSE;
   STATUS[150].EXT.ModeBit3 := FALSE;
   STATUS[150].EXT.BIT19 := FALSE;
   STATUS[150].EXT.BIT20 := FALSE;
   STATUS[150].EXT.AlarmSuppressed := FALSE;
   STATUS[150].EXT.AlarmPresent := FALSE;
   STATUS[150].EXT.AlarmFailUnAck := FALSE;
   STATUS[150].Status := 0;
   STATUS[150].TimeStamp := 16#0000;
   STATUS[151].EXT.AlarmWarnUnAck := FALSE;
   STATUS[151].EXT.AckRequired := FALSE;
   STATUS[151].EXT.Maintanence := FALSE;
   STATUS[151].EXT.Operation := FALSE;
   STATUS[151].EXT.Forced := FALSE;
   STATUS[151].EXT.BIT29 := FALSE;
   STATUS[151].EXT.BIT30 := FALSE;
   STATUS[151].EXT.BIT31 := FALSE;
   STATUS[151].EXT.ModeBit1 := FALSE;
   STATUS[151].EXT.ModeBit2 := FALSE;
   STATUS[151].EXT.ModeBit3 := FALSE;
   STATUS[151].EXT.BIT19 := FALSE;
   STATUS[151].EXT.BIT20 := FALSE;
   STATUS[151].EXT.AlarmSuppressed := FALSE;
   STATUS[151].EXT.AlarmPresent := FALSE;
   STATUS[151].EXT.AlarmFailUnAck := FALSE;
   STATUS[151].Status := 0;
   STATUS[151].TimeStamp := 16#0000;
   STATUS[152].EXT.AlarmWarnUnAck := FALSE;
   STATUS[152].EXT.AckRequired := FALSE;
   STATUS[152].EXT.Maintanence := FALSE;
   STATUS[152].EXT.Operation := FALSE;
   STATUS[152].EXT.Forced := FALSE;
   STATUS[152].EXT.BIT29 := FALSE;
   STATUS[152].EXT.BIT30 := FALSE;
   STATUS[152].EXT.BIT31 := FALSE;
   STATUS[152].EXT.ModeBit1 := FALSE;
   STATUS[152].EXT.ModeBit2 := FALSE;
   STATUS[152].EXT.ModeBit3 := FALSE;
   STATUS[152].EXT.BIT19 := FALSE;
   STATUS[152].EXT.BIT20 := FALSE;
   STATUS[152].EXT.AlarmSuppressed := FALSE;
   STATUS[152].EXT.AlarmPresent := FALSE;
   STATUS[152].EXT.AlarmFailUnAck := FALSE;
   STATUS[152].Status := 0;
   STATUS[152].TimeStamp := 16#0000;
   STATUS[153].EXT.AlarmWarnUnAck := FALSE;
   STATUS[153].EXT.AckRequired := FALSE;
   STATUS[153].EXT.Maintanence := FALSE;
   STATUS[153].EXT.Operation := FALSE;
   STATUS[153].EXT.Forced := FALSE;
   STATUS[153].EXT.BIT29 := FALSE;
   STATUS[153].EXT.BIT30 := FALSE;
   STATUS[153].EXT.BIT31 := FALSE;
   STATUS[153].EXT.ModeBit1 := FALSE;
   STATUS[153].EXT.ModeBit2 := FALSE;
   STATUS[153].EXT.ModeBit3 := FALSE;
   STATUS[153].EXT.BIT19 := FALSE;
   STATUS[153].EXT.BIT20 := FALSE;
   STATUS[153].EXT.AlarmSuppressed := FALSE;
   STATUS[153].EXT.AlarmPresent := FALSE;
   STATUS[153].EXT.AlarmFailUnAck := FALSE;
   STATUS[153].Status := 0;
   STATUS[153].TimeStamp := 16#0000;
   STATUS[154].EXT.AlarmWarnUnAck := FALSE;
   STATUS[154].EXT.AckRequired := FALSE;
   STATUS[154].EXT.Maintanence := FALSE;
   STATUS[154].EXT.Operation := FALSE;
   STATUS[154].EXT.Forced := FALSE;
   STATUS[154].EXT.BIT29 := FALSE;
   STATUS[154].EXT.BIT30 := FALSE;
   STATUS[154].EXT.BIT31 := FALSE;
   STATUS[154].EXT.ModeBit1 := FALSE;
   STATUS[154].EXT.ModeBit2 := FALSE;
   STATUS[154].EXT.ModeBit3 := FALSE;
   STATUS[154].EXT.BIT19 := FALSE;
   STATUS[154].EXT.BIT20 := FALSE;
   STATUS[154].EXT.AlarmSuppressed := FALSE;
   STATUS[154].EXT.AlarmPresent := FALSE;
   STATUS[154].EXT.AlarmFailUnAck := FALSE;
   STATUS[154].Status := 0;
   STATUS[154].TimeStamp := 16#0000;
   STATUS[155].EXT.AlarmWarnUnAck := FALSE;
   STATUS[155].EXT.AckRequired := FALSE;
   STATUS[155].EXT.Maintanence := FALSE;
   STATUS[155].EXT.Operation := FALSE;
   STATUS[155].EXT.Forced := FALSE;
   STATUS[155].EXT.BIT29 := FALSE;
   STATUS[155].EXT.BIT30 := FALSE;
   STATUS[155].EXT.BIT31 := FALSE;
   STATUS[155].EXT.ModeBit1 := FALSE;
   STATUS[155].EXT.ModeBit2 := FALSE;
   STATUS[155].EXT.ModeBit3 := FALSE;
   STATUS[155].EXT.BIT19 := FALSE;
   STATUS[155].EXT.BIT20 := FALSE;
   STATUS[155].EXT.AlarmSuppressed := FALSE;
   STATUS[155].EXT.AlarmPresent := FALSE;
   STATUS[155].EXT.AlarmFailUnAck := FALSE;
   STATUS[155].Status := 0;
   STATUS[155].TimeStamp := 16#0000;
   STATUS[156].EXT.AlarmWarnUnAck := FALSE;
   STATUS[156].EXT.AckRequired := FALSE;
   STATUS[156].EXT.Maintanence := FALSE;
   STATUS[156].EXT.Operation := FALSE;
   STATUS[156].EXT.Forced := FALSE;
   STATUS[156].EXT.BIT29 := FALSE;
   STATUS[156].EXT.BIT30 := FALSE;
   STATUS[156].EXT.BIT31 := FALSE;
   STATUS[156].EXT.ModeBit1 := FALSE;
   STATUS[156].EXT.ModeBit2 := FALSE;
   STATUS[156].EXT.ModeBit3 := FALSE;
   STATUS[156].EXT.BIT19 := FALSE;
   STATUS[156].EXT.BIT20 := FALSE;
   STATUS[156].EXT.AlarmSuppressed := FALSE;
   STATUS[156].EXT.AlarmPresent := FALSE;
   STATUS[156].EXT.AlarmFailUnAck := FALSE;
   STATUS[156].Status := 0;
   STATUS[156].TimeStamp := 16#0000;
   STATUS[157].EXT.AlarmWarnUnAck := FALSE;
   STATUS[157].EXT.AckRequired := FALSE;
   STATUS[157].EXT.Maintanence := FALSE;
   STATUS[157].EXT.Operation := FALSE;
   STATUS[157].EXT.Forced := FALSE;
   STATUS[157].EXT.BIT29 := FALSE;
   STATUS[157].EXT.BIT30 := FALSE;
   STATUS[157].EXT.BIT31 := FALSE;
   STATUS[157].EXT.ModeBit1 := FALSE;
   STATUS[157].EXT.ModeBit2 := FALSE;
   STATUS[157].EXT.ModeBit3 := FALSE;
   STATUS[157].EXT.BIT19 := FALSE;
   STATUS[157].EXT.BIT20 := FALSE;
   STATUS[157].EXT.AlarmSuppressed := FALSE;
   STATUS[157].EXT.AlarmPresent := FALSE;
   STATUS[157].EXT.AlarmFailUnAck := FALSE;
   STATUS[157].Status := 0;
   STATUS[157].TimeStamp := 16#0000;
   STATUS[158].EXT.AlarmWarnUnAck := FALSE;
   STATUS[158].EXT.AckRequired := FALSE;
   STATUS[158].EXT.Maintanence := FALSE;
   STATUS[158].EXT.Operation := FALSE;
   STATUS[158].EXT.Forced := FALSE;
   STATUS[158].EXT.BIT29 := FALSE;
   STATUS[158].EXT.BIT30 := FALSE;
   STATUS[158].EXT.BIT31 := FALSE;
   STATUS[158].EXT.ModeBit1 := FALSE;
   STATUS[158].EXT.ModeBit2 := FALSE;
   STATUS[158].EXT.ModeBit3 := FALSE;
   STATUS[158].EXT.BIT19 := FALSE;
   STATUS[158].EXT.BIT20 := FALSE;
   STATUS[158].EXT.AlarmSuppressed := FALSE;
   STATUS[158].EXT.AlarmPresent := FALSE;
   STATUS[158].EXT.AlarmFailUnAck := FALSE;
   STATUS[158].Status := 0;
   STATUS[158].TimeStamp := 16#0000;
   STATUS[159].EXT.AlarmWarnUnAck := FALSE;
   STATUS[159].EXT.AckRequired := FALSE;
   STATUS[159].EXT.Maintanence := FALSE;
   STATUS[159].EXT.Operation := FALSE;
   STATUS[159].EXT.Forced := FALSE;
   STATUS[159].EXT.BIT29 := FALSE;
   STATUS[159].EXT.BIT30 := FALSE;
   STATUS[159].EXT.BIT31 := FALSE;
   STATUS[159].EXT.ModeBit1 := FALSE;
   STATUS[159].EXT.ModeBit2 := FALSE;
   STATUS[159].EXT.ModeBit3 := FALSE;
   STATUS[159].EXT.BIT19 := FALSE;
   STATUS[159].EXT.BIT20 := FALSE;
   STATUS[159].EXT.AlarmSuppressed := FALSE;
   STATUS[159].EXT.AlarmPresent := FALSE;
   STATUS[159].EXT.AlarmFailUnAck := FALSE;
   STATUS[159].Status := 0;
   STATUS[159].TimeStamp := 16#0000;
   STATUS[160].EXT.AlarmWarnUnAck := FALSE;
   STATUS[160].EXT.AckRequired := FALSE;
   STATUS[160].EXT.Maintanence := FALSE;
   STATUS[160].EXT.Operation := FALSE;
   STATUS[160].EXT.Forced := FALSE;
   STATUS[160].EXT.BIT29 := FALSE;
   STATUS[160].EXT.BIT30 := FALSE;
   STATUS[160].EXT.BIT31 := FALSE;
   STATUS[160].EXT.ModeBit1 := FALSE;
   STATUS[160].EXT.ModeBit2 := FALSE;
   STATUS[160].EXT.ModeBit3 := FALSE;
   STATUS[160].EXT.BIT19 := FALSE;
   STATUS[160].EXT.BIT20 := FALSE;
   STATUS[160].EXT.AlarmSuppressed := FALSE;
   STATUS[160].EXT.AlarmPresent := FALSE;
   STATUS[160].EXT.AlarmFailUnAck := FALSE;
   STATUS[160].Status := 0;
   STATUS[160].TimeStamp := 16#0000;
   STATUS[161].EXT.AlarmWarnUnAck := FALSE;
   STATUS[161].EXT.AckRequired := FALSE;
   STATUS[161].EXT.Maintanence := FALSE;
   STATUS[161].EXT.Operation := FALSE;
   STATUS[161].EXT.Forced := FALSE;
   STATUS[161].EXT.BIT29 := FALSE;
   STATUS[161].EXT.BIT30 := FALSE;
   STATUS[161].EXT.BIT31 := FALSE;
   STATUS[161].EXT.ModeBit1 := FALSE;
   STATUS[161].EXT.ModeBit2 := FALSE;
   STATUS[161].EXT.ModeBit3 := FALSE;
   STATUS[161].EXT.BIT19 := FALSE;
   STATUS[161].EXT.BIT20 := FALSE;
   STATUS[161].EXT.AlarmSuppressed := FALSE;
   STATUS[161].EXT.AlarmPresent := FALSE;
   STATUS[161].EXT.AlarmFailUnAck := FALSE;
   STATUS[161].Status := 0;
   STATUS[161].TimeStamp := 16#0000;
   STATUS[162].EXT.AlarmWarnUnAck := FALSE;
   STATUS[162].EXT.AckRequired := FALSE;
   STATUS[162].EXT.Maintanence := FALSE;
   STATUS[162].EXT.Operation := FALSE;
   STATUS[162].EXT.Forced := FALSE;
   STATUS[162].EXT.BIT29 := FALSE;
   STATUS[162].EXT.BIT30 := FALSE;
   STATUS[162].EXT.BIT31 := FALSE;
   STATUS[162].EXT.ModeBit1 := FALSE;
   STATUS[162].EXT.ModeBit2 := FALSE;
   STATUS[162].EXT.ModeBit3 := FALSE;
   STATUS[162].EXT.BIT19 := FALSE;
   STATUS[162].EXT.BIT20 := FALSE;
   STATUS[162].EXT.AlarmSuppressed := FALSE;
   STATUS[162].EXT.AlarmPresent := FALSE;
   STATUS[162].EXT.AlarmFailUnAck := FALSE;
   STATUS[162].Status := 0;
   STATUS[162].TimeStamp := 16#0000;
   STATUS[163].EXT.AlarmWarnUnAck := FALSE;
   STATUS[163].EXT.AckRequired := FALSE;
   STATUS[163].EXT.Maintanence := FALSE;
   STATUS[163].EXT.Operation := FALSE;
   STATUS[163].EXT.Forced := FALSE;
   STATUS[163].EXT.BIT29 := FALSE;
   STATUS[163].EXT.BIT30 := FALSE;
   STATUS[163].EXT.BIT31 := FALSE;
   STATUS[163].EXT.ModeBit1 := FALSE;
   STATUS[163].EXT.ModeBit2 := FALSE;
   STATUS[163].EXT.ModeBit3 := FALSE;
   STATUS[163].EXT.BIT19 := FALSE;
   STATUS[163].EXT.BIT20 := FALSE;
   STATUS[163].EXT.AlarmSuppressed := FALSE;
   STATUS[163].EXT.AlarmPresent := FALSE;
   STATUS[163].EXT.AlarmFailUnAck := FALSE;
   STATUS[163].Status := 0;
   STATUS[163].TimeStamp := 16#0000;
   STATUS[164].EXT.AlarmWarnUnAck := FALSE;
   STATUS[164].EXT.AckRequired := FALSE;
   STATUS[164].EXT.Maintanence := FALSE;
   STATUS[164].EXT.Operation := FALSE;
   STATUS[164].EXT.Forced := FALSE;
   STATUS[164].EXT.BIT29 := FALSE;
   STATUS[164].EXT.BIT30 := FALSE;
   STATUS[164].EXT.BIT31 := FALSE;
   STATUS[164].EXT.ModeBit1 := FALSE;
   STATUS[164].EXT.ModeBit2 := FALSE;
   STATUS[164].EXT.ModeBit3 := FALSE;
   STATUS[164].EXT.BIT19 := FALSE;
   STATUS[164].EXT.BIT20 := FALSE;
   STATUS[164].EXT.AlarmSuppressed := FALSE;
   STATUS[164].EXT.AlarmPresent := FALSE;
   STATUS[164].EXT.AlarmFailUnAck := FALSE;
   STATUS[164].Status := 0;
   STATUS[164].TimeStamp := 16#0000;
   STATUS[165].EXT.AlarmWarnUnAck := FALSE;
   STATUS[165].EXT.AckRequired := FALSE;
   STATUS[165].EXT.Maintanence := FALSE;
   STATUS[165].EXT.Operation := FALSE;
   STATUS[165].EXT.Forced := FALSE;
   STATUS[165].EXT.BIT29 := FALSE;
   STATUS[165].EXT.BIT30 := FALSE;
   STATUS[165].EXT.BIT31 := FALSE;
   STATUS[165].EXT.ModeBit1 := FALSE;
   STATUS[165].EXT.ModeBit2 := FALSE;
   STATUS[165].EXT.ModeBit3 := FALSE;
   STATUS[165].EXT.BIT19 := FALSE;
   STATUS[165].EXT.BIT20 := FALSE;
   STATUS[165].EXT.AlarmSuppressed := FALSE;
   STATUS[165].EXT.AlarmPresent := FALSE;
   STATUS[165].EXT.AlarmFailUnAck := FALSE;
   STATUS[165].Status := 0;
   STATUS[165].TimeStamp := 16#0000;
   STATUS[166].EXT.AlarmWarnUnAck := FALSE;
   STATUS[166].EXT.AckRequired := FALSE;
   STATUS[166].EXT.Maintanence := FALSE;
   STATUS[166].EXT.Operation := FALSE;
   STATUS[166].EXT.Forced := FALSE;
   STATUS[166].EXT.BIT29 := FALSE;
   STATUS[166].EXT.BIT30 := FALSE;
   STATUS[166].EXT.BIT31 := FALSE;
   STATUS[166].EXT.ModeBit1 := FALSE;
   STATUS[166].EXT.ModeBit2 := FALSE;
   STATUS[166].EXT.ModeBit3 := FALSE;
   STATUS[166].EXT.BIT19 := FALSE;
   STATUS[166].EXT.BIT20 := FALSE;
   STATUS[166].EXT.AlarmSuppressed := FALSE;
   STATUS[166].EXT.AlarmPresent := FALSE;
   STATUS[166].EXT.AlarmFailUnAck := FALSE;
   STATUS[166].Status := 0;
   STATUS[166].TimeStamp := 16#0000;
   STATUS[167].EXT.AlarmWarnUnAck := FALSE;
   STATUS[167].EXT.AckRequired := FALSE;
   STATUS[167].EXT.Maintanence := FALSE;
   STATUS[167].EXT.Operation := FALSE;
   STATUS[167].EXT.Forced := FALSE;
   STATUS[167].EXT.BIT29 := FALSE;
   STATUS[167].EXT.BIT30 := FALSE;
   STATUS[167].EXT.BIT31 := FALSE;
   STATUS[167].EXT.ModeBit1 := FALSE;
   STATUS[167].EXT.ModeBit2 := FALSE;
   STATUS[167].EXT.ModeBit3 := FALSE;
   STATUS[167].EXT.BIT19 := FALSE;
   STATUS[167].EXT.BIT20 := FALSE;
   STATUS[167].EXT.AlarmSuppressed := FALSE;
   STATUS[167].EXT.AlarmPresent := FALSE;
   STATUS[167].EXT.AlarmFailUnAck := FALSE;
   STATUS[167].Status := 0;
   STATUS[167].TimeStamp := 16#0000;
   STATUS[168].EXT.AlarmWarnUnAck := FALSE;
   STATUS[168].EXT.AckRequired := FALSE;
   STATUS[168].EXT.Maintanence := FALSE;
   STATUS[168].EXT.Operation := FALSE;
   STATUS[168].EXT.Forced := FALSE;
   STATUS[168].EXT.BIT29 := FALSE;
   STATUS[168].EXT.BIT30 := FALSE;
   STATUS[168].EXT.BIT31 := FALSE;
   STATUS[168].EXT.ModeBit1 := FALSE;
   STATUS[168].EXT.ModeBit2 := FALSE;
   STATUS[168].EXT.ModeBit3 := FALSE;
   STATUS[168].EXT.BIT19 := FALSE;
   STATUS[168].EXT.BIT20 := FALSE;
   STATUS[168].EXT.AlarmSuppressed := FALSE;
   STATUS[168].EXT.AlarmPresent := FALSE;
   STATUS[168].EXT.AlarmFailUnAck := FALSE;
   STATUS[168].Status := 0;
   STATUS[168].TimeStamp := 16#0000;
   STATUS[169].EXT.AlarmWarnUnAck := FALSE;
   STATUS[169].EXT.AckRequired := FALSE;
   STATUS[169].EXT.Maintanence := FALSE;
   STATUS[169].EXT.Operation := FALSE;
   STATUS[169].EXT.Forced := FALSE;
   STATUS[169].EXT.BIT29 := FALSE;
   STATUS[169].EXT.BIT30 := FALSE;
   STATUS[169].EXT.BIT31 := FALSE;
   STATUS[169].EXT.ModeBit1 := FALSE;
   STATUS[169].EXT.ModeBit2 := FALSE;
   STATUS[169].EXT.ModeBit3 := FALSE;
   STATUS[169].EXT.BIT19 := FALSE;
   STATUS[169].EXT.BIT20 := FALSE;
   STATUS[169].EXT.AlarmSuppressed := FALSE;
   STATUS[169].EXT.AlarmPresent := FALSE;
   STATUS[169].EXT.AlarmFailUnAck := FALSE;
   STATUS[169].Status := 0;
   STATUS[169].TimeStamp := 16#0000;
   STATUS[170].EXT.AlarmWarnUnAck := FALSE;
   STATUS[170].EXT.AckRequired := FALSE;
   STATUS[170].EXT.Maintanence := FALSE;
   STATUS[170].EXT.Operation := FALSE;
   STATUS[170].EXT.Forced := FALSE;
   STATUS[170].EXT.BIT29 := FALSE;
   STATUS[170].EXT.BIT30 := FALSE;
   STATUS[170].EXT.BIT31 := FALSE;
   STATUS[170].EXT.ModeBit1 := FALSE;
   STATUS[170].EXT.ModeBit2 := FALSE;
   STATUS[170].EXT.ModeBit3 := FALSE;
   STATUS[170].EXT.BIT19 := FALSE;
   STATUS[170].EXT.BIT20 := FALSE;
   STATUS[170].EXT.AlarmSuppressed := FALSE;
   STATUS[170].EXT.AlarmPresent := FALSE;
   STATUS[170].EXT.AlarmFailUnAck := FALSE;
   STATUS[170].Status := -22466;
   STATUS[170].TimeStamp := 16#84BA;
   STATUS[171].EXT.AlarmWarnUnAck := FALSE;
   STATUS[171].EXT.AckRequired := FALSE;
   STATUS[171].EXT.Maintanence := FALSE;
   STATUS[171].EXT.Operation := FALSE;
   STATUS[171].EXT.Forced := FALSE;
   STATUS[171].EXT.BIT29 := FALSE;
   STATUS[171].EXT.BIT30 := FALSE;
   STATUS[171].EXT.BIT31 := FALSE;
   STATUS[171].EXT.ModeBit1 := FALSE;
   STATUS[171].EXT.ModeBit2 := FALSE;
   STATUS[171].EXT.ModeBit3 := FALSE;
   STATUS[171].EXT.BIT19 := FALSE;
   STATUS[171].EXT.BIT20 := FALSE;
   STATUS[171].EXT.AlarmSuppressed := FALSE;
   STATUS[171].EXT.AlarmPresent := FALSE;
   STATUS[171].EXT.AlarmFailUnAck := FALSE;
   STATUS[171].Status := 0;
   STATUS[171].TimeStamp := 16#0000;
   STATUS[172].EXT.AlarmWarnUnAck := FALSE;
   STATUS[172].EXT.AckRequired := FALSE;
   STATUS[172].EXT.Maintanence := FALSE;
   STATUS[172].EXT.Operation := FALSE;
   STATUS[172].EXT.Forced := FALSE;
   STATUS[172].EXT.BIT29 := FALSE;
   STATUS[172].EXT.BIT30 := FALSE;
   STATUS[172].EXT.BIT31 := FALSE;
   STATUS[172].EXT.ModeBit1 := FALSE;
   STATUS[172].EXT.ModeBit2 := FALSE;
   STATUS[172].EXT.ModeBit3 := FALSE;
   STATUS[172].EXT.BIT19 := FALSE;
   STATUS[172].EXT.BIT20 := FALSE;
   STATUS[172].EXT.AlarmSuppressed := FALSE;
   STATUS[172].EXT.AlarmPresent := FALSE;
   STATUS[172].EXT.AlarmFailUnAck := FALSE;
   STATUS[172].Status := 0;
   STATUS[172].TimeStamp := 16#0000;
   STATUS[173].EXT.AlarmWarnUnAck := FALSE;
   STATUS[173].EXT.AckRequired := FALSE;
   STATUS[173].EXT.Maintanence := FALSE;
   STATUS[173].EXT.Operation := FALSE;
   STATUS[173].EXT.Forced := FALSE;
   STATUS[173].EXT.BIT29 := FALSE;
   STATUS[173].EXT.BIT30 := FALSE;
   STATUS[173].EXT.BIT31 := FALSE;
   STATUS[173].EXT.ModeBit1 := FALSE;
   STATUS[173].EXT.ModeBit2 := FALSE;
   STATUS[173].EXT.ModeBit3 := FALSE;
   STATUS[173].EXT.BIT19 := FALSE;
   STATUS[173].EXT.BIT20 := FALSE;
   STATUS[173].EXT.AlarmSuppressed := FALSE;
   STATUS[173].EXT.AlarmPresent := FALSE;
   STATUS[173].EXT.AlarmFailUnAck := FALSE;
   STATUS[173].Status := 0;
   STATUS[173].TimeStamp := 16#0000;
   STATUS[174].EXT.AlarmWarnUnAck := FALSE;
   STATUS[174].EXT.AckRequired := FALSE;
   STATUS[174].EXT.Maintanence := FALSE;
   STATUS[174].EXT.Operation := FALSE;
   STATUS[174].EXT.Forced := FALSE;
   STATUS[174].EXT.BIT29 := FALSE;
   STATUS[174].EXT.BIT30 := FALSE;
   STATUS[174].EXT.BIT31 := FALSE;
   STATUS[174].EXT.ModeBit1 := FALSE;
   STATUS[174].EXT.ModeBit2 := FALSE;
   STATUS[174].EXT.ModeBit3 := FALSE;
   STATUS[174].EXT.BIT19 := FALSE;
   STATUS[174].EXT.BIT20 := FALSE;
   STATUS[174].EXT.AlarmSuppressed := FALSE;
   STATUS[174].EXT.AlarmPresent := FALSE;
   STATUS[174].EXT.AlarmFailUnAck := FALSE;
   STATUS[174].Status := 0;
   STATUS[174].TimeStamp := 16#0000;
   STATUS[175].EXT.AlarmWarnUnAck := FALSE;
   STATUS[175].EXT.AckRequired := FALSE;
   STATUS[175].EXT.Maintanence := FALSE;
   STATUS[175].EXT.Operation := FALSE;
   STATUS[175].EXT.Forced := FALSE;
   STATUS[175].EXT.BIT29 := FALSE;
   STATUS[175].EXT.BIT30 := FALSE;
   STATUS[175].EXT.BIT31 := FALSE;
   STATUS[175].EXT.ModeBit1 := FALSE;
   STATUS[175].EXT.ModeBit2 := FALSE;
   STATUS[175].EXT.ModeBit3 := FALSE;
   STATUS[175].EXT.BIT19 := FALSE;
   STATUS[175].EXT.BIT20 := FALSE;
   STATUS[175].EXT.AlarmSuppressed := FALSE;
   STATUS[175].EXT.AlarmPresent := FALSE;
   STATUS[175].EXT.AlarmFailUnAck := FALSE;
   STATUS[175].Status := 0;
   STATUS[175].TimeStamp := 16#0000;
   STATUS[176].EXT.AlarmWarnUnAck := FALSE;
   STATUS[176].EXT.AckRequired := FALSE;
   STATUS[176].EXT.Maintanence := FALSE;
   STATUS[176].EXT.Operation := FALSE;
   STATUS[176].EXT.Forced := FALSE;
   STATUS[176].EXT.BIT29 := FALSE;
   STATUS[176].EXT.BIT30 := FALSE;
   STATUS[176].EXT.BIT31 := FALSE;
   STATUS[176].EXT.ModeBit1 := FALSE;
   STATUS[176].EXT.ModeBit2 := FALSE;
   STATUS[176].EXT.ModeBit3 := FALSE;
   STATUS[176].EXT.BIT19 := FALSE;
   STATUS[176].EXT.BIT20 := FALSE;
   STATUS[176].EXT.AlarmSuppressed := FALSE;
   STATUS[176].EXT.AlarmPresent := FALSE;
   STATUS[176].EXT.AlarmFailUnAck := FALSE;
   STATUS[176].Status := 0;
   STATUS[176].TimeStamp := 16#0000;
   STATUS[177].EXT.AlarmWarnUnAck := FALSE;
   STATUS[177].EXT.AckRequired := FALSE;
   STATUS[177].EXT.Maintanence := FALSE;
   STATUS[177].EXT.Operation := FALSE;
   STATUS[177].EXT.Forced := FALSE;
   STATUS[177].EXT.BIT29 := FALSE;
   STATUS[177].EXT.BIT30 := FALSE;
   STATUS[177].EXT.BIT31 := FALSE;
   STATUS[177].EXT.ModeBit1 := FALSE;
   STATUS[177].EXT.ModeBit2 := FALSE;
   STATUS[177].EXT.ModeBit3 := FALSE;
   STATUS[177].EXT.BIT19 := FALSE;
   STATUS[177].EXT.BIT20 := FALSE;
   STATUS[177].EXT.AlarmSuppressed := FALSE;
   STATUS[177].EXT.AlarmPresent := FALSE;
   STATUS[177].EXT.AlarmFailUnAck := FALSE;
   STATUS[177].Status := 0;
   STATUS[177].TimeStamp := 16#0000;
   STATUS[178].EXT.AlarmWarnUnAck := FALSE;
   STATUS[178].EXT.AckRequired := FALSE;
   STATUS[178].EXT.Maintanence := FALSE;
   STATUS[178].EXT.Operation := FALSE;
   STATUS[178].EXT.Forced := FALSE;
   STATUS[178].EXT.BIT29 := FALSE;
   STATUS[178].EXT.BIT30 := FALSE;
   STATUS[178].EXT.BIT31 := FALSE;
   STATUS[178].EXT.ModeBit1 := FALSE;
   STATUS[178].EXT.ModeBit2 := FALSE;
   STATUS[178].EXT.ModeBit3 := FALSE;
   STATUS[178].EXT.BIT19 := FALSE;
   STATUS[178].EXT.BIT20 := FALSE;
   STATUS[178].EXT.AlarmSuppressed := FALSE;
   STATUS[178].EXT.AlarmPresent := FALSE;
   STATUS[178].EXT.AlarmFailUnAck := FALSE;
   STATUS[178].Status := 0;
   STATUS[178].TimeStamp := 16#0000;
   STATUS[179].EXT.AlarmWarnUnAck := FALSE;
   STATUS[179].EXT.AckRequired := FALSE;
   STATUS[179].EXT.Maintanence := FALSE;
   STATUS[179].EXT.Operation := FALSE;
   STATUS[179].EXT.Forced := FALSE;
   STATUS[179].EXT.BIT29 := FALSE;
   STATUS[179].EXT.BIT30 := FALSE;
   STATUS[179].EXT.BIT31 := FALSE;
   STATUS[179].EXT.ModeBit1 := FALSE;
   STATUS[179].EXT.ModeBit2 := FALSE;
   STATUS[179].EXT.ModeBit3 := FALSE;
   STATUS[179].EXT.BIT19 := FALSE;
   STATUS[179].EXT.BIT20 := FALSE;
   STATUS[179].EXT.AlarmSuppressed := FALSE;
   STATUS[179].EXT.AlarmPresent := FALSE;
   STATUS[179].EXT.AlarmFailUnAck := FALSE;
   STATUS[179].Status := 0;
   STATUS[179].TimeStamp := 16#0000;
   STATUS[180].EXT.AlarmWarnUnAck := FALSE;
   STATUS[180].EXT.AckRequired := FALSE;
   STATUS[180].EXT.Maintanence := FALSE;
   STATUS[180].EXT.Operation := FALSE;
   STATUS[180].EXT.Forced := FALSE;
   STATUS[180].EXT.BIT29 := FALSE;
   STATUS[180].EXT.BIT30 := FALSE;
   STATUS[180].EXT.BIT31 := FALSE;
   STATUS[180].EXT.ModeBit1 := FALSE;
   STATUS[180].EXT.ModeBit2 := FALSE;
   STATUS[180].EXT.ModeBit3 := FALSE;
   STATUS[180].EXT.BIT19 := FALSE;
   STATUS[180].EXT.BIT20 := FALSE;
   STATUS[180].EXT.AlarmSuppressed := FALSE;
   STATUS[180].EXT.AlarmPresent := FALSE;
   STATUS[180].EXT.AlarmFailUnAck := FALSE;
   STATUS[180].Status := 0;
   STATUS[180].TimeStamp := 16#0000;
   STATUS[181].EXT.AlarmWarnUnAck := FALSE;
   STATUS[181].EXT.AckRequired := FALSE;
   STATUS[181].EXT.Maintanence := FALSE;
   STATUS[181].EXT.Operation := FALSE;
   STATUS[181].EXT.Forced := FALSE;
   STATUS[181].EXT.BIT29 := FALSE;
   STATUS[181].EXT.BIT30 := FALSE;
   STATUS[181].EXT.BIT31 := FALSE;
   STATUS[181].EXT.ModeBit1 := FALSE;
   STATUS[181].EXT.ModeBit2 := FALSE;
   STATUS[181].EXT.ModeBit3 := FALSE;
   STATUS[181].EXT.BIT19 := FALSE;
   STATUS[181].EXT.BIT20 := FALSE;
   STATUS[181].EXT.AlarmSuppressed := FALSE;
   STATUS[181].EXT.AlarmPresent := FALSE;
   STATUS[181].EXT.AlarmFailUnAck := FALSE;
   STATUS[181].Status := 0;
   STATUS[181].TimeStamp := 16#0000;
   STATUS[182].EXT.AlarmWarnUnAck := FALSE;
   STATUS[182].EXT.AckRequired := FALSE;
   STATUS[182].EXT.Maintanence := FALSE;
   STATUS[182].EXT.Operation := FALSE;
   STATUS[182].EXT.Forced := FALSE;
   STATUS[182].EXT.BIT29 := FALSE;
   STATUS[182].EXT.BIT30 := FALSE;
   STATUS[182].EXT.BIT31 := FALSE;
   STATUS[182].EXT.ModeBit1 := FALSE;
   STATUS[182].EXT.ModeBit2 := FALSE;
   STATUS[182].EXT.ModeBit3 := FALSE;
   STATUS[182].EXT.BIT19 := FALSE;
   STATUS[182].EXT.BIT20 := FALSE;
   STATUS[182].EXT.AlarmSuppressed := FALSE;
   STATUS[182].EXT.AlarmPresent := FALSE;
   STATUS[182].EXT.AlarmFailUnAck := FALSE;
   STATUS[182].Status := 0;
   STATUS[182].TimeStamp := 16#0000;
   STATUS[183].EXT.AlarmWarnUnAck := FALSE;
   STATUS[183].EXT.AckRequired := FALSE;
   STATUS[183].EXT.Maintanence := FALSE;
   STATUS[183].EXT.Operation := FALSE;
   STATUS[183].EXT.Forced := FALSE;
   STATUS[183].EXT.BIT29 := FALSE;
   STATUS[183].EXT.BIT30 := FALSE;
   STATUS[183].EXT.BIT31 := FALSE;
   STATUS[183].EXT.ModeBit1 := FALSE;
   STATUS[183].EXT.ModeBit2 := FALSE;
   STATUS[183].EXT.ModeBit3 := FALSE;
   STATUS[183].EXT.BIT19 := FALSE;
   STATUS[183].EXT.BIT20 := FALSE;
   STATUS[183].EXT.AlarmSuppressed := FALSE;
   STATUS[183].EXT.AlarmPresent := FALSE;
   STATUS[183].EXT.AlarmFailUnAck := FALSE;
   STATUS[183].Status := 0;
   STATUS[183].TimeStamp := 16#0000;
   STATUS[184].EXT.AlarmWarnUnAck := FALSE;
   STATUS[184].EXT.AckRequired := FALSE;
   STATUS[184].EXT.Maintanence := FALSE;
   STATUS[184].EXT.Operation := FALSE;
   STATUS[184].EXT.Forced := FALSE;
   STATUS[184].EXT.BIT29 := FALSE;
   STATUS[184].EXT.BIT30 := FALSE;
   STATUS[184].EXT.BIT31 := FALSE;
   STATUS[184].EXT.ModeBit1 := FALSE;
   STATUS[184].EXT.ModeBit2 := FALSE;
   STATUS[184].EXT.ModeBit3 := FALSE;
   STATUS[184].EXT.BIT19 := FALSE;
   STATUS[184].EXT.BIT20 := FALSE;
   STATUS[184].EXT.AlarmSuppressed := FALSE;
   STATUS[184].EXT.AlarmPresent := FALSE;
   STATUS[184].EXT.AlarmFailUnAck := FALSE;
   STATUS[184].Status := 0;
   STATUS[184].TimeStamp := 16#0000;
   STATUS[185].EXT.AlarmWarnUnAck := FALSE;
   STATUS[185].EXT.AckRequired := FALSE;
   STATUS[185].EXT.Maintanence := FALSE;
   STATUS[185].EXT.Operation := FALSE;
   STATUS[185].EXT.Forced := FALSE;
   STATUS[185].EXT.BIT29 := FALSE;
   STATUS[185].EXT.BIT30 := FALSE;
   STATUS[185].EXT.BIT31 := FALSE;
   STATUS[185].EXT.ModeBit1 := FALSE;
   STATUS[185].EXT.ModeBit2 := FALSE;
   STATUS[185].EXT.ModeBit3 := FALSE;
   STATUS[185].EXT.BIT19 := FALSE;
   STATUS[185].EXT.BIT20 := FALSE;
   STATUS[185].EXT.AlarmSuppressed := FALSE;
   STATUS[185].EXT.AlarmPresent := FALSE;
   STATUS[185].EXT.AlarmFailUnAck := FALSE;
   STATUS[185].Status := 0;
   STATUS[185].TimeStamp := 16#0000;
   STATUS[186].EXT.AlarmWarnUnAck := FALSE;
   STATUS[186].EXT.AckRequired := FALSE;
   STATUS[186].EXT.Maintanence := FALSE;
   STATUS[186].EXT.Operation := FALSE;
   STATUS[186].EXT.Forced := FALSE;
   STATUS[186].EXT.BIT29 := FALSE;
   STATUS[186].EXT.BIT30 := FALSE;
   STATUS[186].EXT.BIT31 := FALSE;
   STATUS[186].EXT.ModeBit1 := FALSE;
   STATUS[186].EXT.ModeBit2 := FALSE;
   STATUS[186].EXT.ModeBit3 := FALSE;
   STATUS[186].EXT.BIT19 := FALSE;
   STATUS[186].EXT.BIT20 := FALSE;
   STATUS[186].EXT.AlarmSuppressed := FALSE;
   STATUS[186].EXT.AlarmPresent := FALSE;
   STATUS[186].EXT.AlarmFailUnAck := FALSE;
   STATUS[186].Status := 0;
   STATUS[186].TimeStamp := 16#0000;
   STATUS[187].EXT.AlarmWarnUnAck := FALSE;
   STATUS[187].EXT.AckRequired := FALSE;
   STATUS[187].EXT.Maintanence := FALSE;
   STATUS[187].EXT.Operation := FALSE;
   STATUS[187].EXT.Forced := FALSE;
   STATUS[187].EXT.BIT29 := FALSE;
   STATUS[187].EXT.BIT30 := FALSE;
   STATUS[187].EXT.BIT31 := FALSE;
   STATUS[187].EXT.ModeBit1 := FALSE;
   STATUS[187].EXT.ModeBit2 := FALSE;
   STATUS[187].EXT.ModeBit3 := FALSE;
   STATUS[187].EXT.BIT19 := FALSE;
   STATUS[187].EXT.BIT20 := FALSE;
   STATUS[187].EXT.AlarmSuppressed := FALSE;
   STATUS[187].EXT.AlarmPresent := FALSE;
   STATUS[187].EXT.AlarmFailUnAck := FALSE;
   STATUS[187].Status := 0;
   STATUS[187].TimeStamp := 16#0000;
   STATUS[188].EXT.AlarmWarnUnAck := FALSE;
   STATUS[188].EXT.AckRequired := FALSE;
   STATUS[188].EXT.Maintanence := FALSE;
   STATUS[188].EXT.Operation := FALSE;
   STATUS[188].EXT.Forced := FALSE;
   STATUS[188].EXT.BIT29 := FALSE;
   STATUS[188].EXT.BIT30 := FALSE;
   STATUS[188].EXT.BIT31 := FALSE;
   STATUS[188].EXT.ModeBit1 := FALSE;
   STATUS[188].EXT.ModeBit2 := FALSE;
   STATUS[188].EXT.ModeBit3 := FALSE;
   STATUS[188].EXT.BIT19 := FALSE;
   STATUS[188].EXT.BIT20 := FALSE;
   STATUS[188].EXT.AlarmSuppressed := FALSE;
   STATUS[188].EXT.AlarmPresent := FALSE;
   STATUS[188].EXT.AlarmFailUnAck := FALSE;
   STATUS[188].Status := 0;
   STATUS[188].TimeStamp := 16#0000;
   STATUS[189].EXT.AlarmWarnUnAck := FALSE;
   STATUS[189].EXT.AckRequired := FALSE;
   STATUS[189].EXT.Maintanence := FALSE;
   STATUS[189].EXT.Operation := FALSE;
   STATUS[189].EXT.Forced := FALSE;
   STATUS[189].EXT.BIT29 := FALSE;
   STATUS[189].EXT.BIT30 := FALSE;
   STATUS[189].EXT.BIT31 := FALSE;
   STATUS[189].EXT.ModeBit1 := FALSE;
   STATUS[189].EXT.ModeBit2 := FALSE;
   STATUS[189].EXT.ModeBit3 := FALSE;
   STATUS[189].EXT.BIT19 := FALSE;
   STATUS[189].EXT.BIT20 := FALSE;
   STATUS[189].EXT.AlarmSuppressed := FALSE;
   STATUS[189].EXT.AlarmPresent := FALSE;
   STATUS[189].EXT.AlarmFailUnAck := FALSE;
   STATUS[189].Status := 0;
   STATUS[189].TimeStamp := 16#0000;
   STATUS[190].EXT.AlarmWarnUnAck := FALSE;
   STATUS[190].EXT.AckRequired := FALSE;
   STATUS[190].EXT.Maintanence := FALSE;
   STATUS[190].EXT.Operation := FALSE;
   STATUS[190].EXT.Forced := FALSE;
   STATUS[190].EXT.BIT29 := FALSE;
   STATUS[190].EXT.BIT30 := FALSE;
   STATUS[190].EXT.BIT31 := FALSE;
   STATUS[190].EXT.ModeBit1 := FALSE;
   STATUS[190].EXT.ModeBit2 := FALSE;
   STATUS[190].EXT.ModeBit3 := FALSE;
   STATUS[190].EXT.BIT19 := FALSE;
   STATUS[190].EXT.BIT20 := FALSE;
   STATUS[190].EXT.AlarmSuppressed := FALSE;
   STATUS[190].EXT.AlarmPresent := FALSE;
   STATUS[190].EXT.AlarmFailUnAck := FALSE;
   STATUS[190].Status := 0;
   STATUS[190].TimeStamp := 16#0000;
   STATUS[191].EXT.AlarmWarnUnAck := FALSE;
   STATUS[191].EXT.AckRequired := FALSE;
   STATUS[191].EXT.Maintanence := FALSE;
   STATUS[191].EXT.Operation := FALSE;
   STATUS[191].EXT.Forced := FALSE;
   STATUS[191].EXT.BIT29 := FALSE;
   STATUS[191].EXT.BIT30 := FALSE;
   STATUS[191].EXT.BIT31 := FALSE;
   STATUS[191].EXT.ModeBit1 := FALSE;
   STATUS[191].EXT.ModeBit2 := FALSE;
   STATUS[191].EXT.ModeBit3 := FALSE;
   STATUS[191].EXT.BIT19 := FALSE;
   STATUS[191].EXT.BIT20 := FALSE;
   STATUS[191].EXT.AlarmSuppressed := FALSE;
   STATUS[191].EXT.AlarmPresent := FALSE;
   STATUS[191].EXT.AlarmFailUnAck := FALSE;
   STATUS[191].Status := 0;
   STATUS[191].TimeStamp := 16#0000;
   STATUS[192].EXT.AlarmWarnUnAck := FALSE;
   STATUS[192].EXT.AckRequired := FALSE;
   STATUS[192].EXT.Maintanence := FALSE;
   STATUS[192].EXT.Operation := FALSE;
   STATUS[192].EXT.Forced := FALSE;
   STATUS[192].EXT.BIT29 := FALSE;
   STATUS[192].EXT.BIT30 := FALSE;
   STATUS[192].EXT.BIT31 := FALSE;
   STATUS[192].EXT.ModeBit1 := FALSE;
   STATUS[192].EXT.ModeBit2 := FALSE;
   STATUS[192].EXT.ModeBit3 := FALSE;
   STATUS[192].EXT.BIT19 := FALSE;
   STATUS[192].EXT.BIT20 := FALSE;
   STATUS[192].EXT.AlarmSuppressed := FALSE;
   STATUS[192].EXT.AlarmPresent := FALSE;
   STATUS[192].EXT.AlarmFailUnAck := FALSE;
   STATUS[192].Status := 0;
   STATUS[192].TimeStamp := 16#0000;
   STATUS[193].EXT.AlarmWarnUnAck := FALSE;
   STATUS[193].EXT.AckRequired := FALSE;
   STATUS[193].EXT.Maintanence := FALSE;
   STATUS[193].EXT.Operation := FALSE;
   STATUS[193].EXT.Forced := FALSE;
   STATUS[193].EXT.BIT29 := FALSE;
   STATUS[193].EXT.BIT30 := FALSE;
   STATUS[193].EXT.BIT31 := FALSE;
   STATUS[193].EXT.ModeBit1 := FALSE;
   STATUS[193].EXT.ModeBit2 := FALSE;
   STATUS[193].EXT.ModeBit3 := FALSE;
   STATUS[193].EXT.BIT19 := FALSE;
   STATUS[193].EXT.BIT20 := FALSE;
   STATUS[193].EXT.AlarmSuppressed := FALSE;
   STATUS[193].EXT.AlarmPresent := FALSE;
   STATUS[193].EXT.AlarmFailUnAck := FALSE;
   STATUS[193].Status := 0;
   STATUS[193].TimeStamp := 16#0000;
   STATUS[194].EXT.AlarmWarnUnAck := FALSE;
   STATUS[194].EXT.AckRequired := FALSE;
   STATUS[194].EXT.Maintanence := FALSE;
   STATUS[194].EXT.Operation := FALSE;
   STATUS[194].EXT.Forced := FALSE;
   STATUS[194].EXT.BIT29 := FALSE;
   STATUS[194].EXT.BIT30 := FALSE;
   STATUS[194].EXT.BIT31 := FALSE;
   STATUS[194].EXT.ModeBit1 := FALSE;
   STATUS[194].EXT.ModeBit2 := FALSE;
   STATUS[194].EXT.ModeBit3 := FALSE;
   STATUS[194].EXT.BIT19 := FALSE;
   STATUS[194].EXT.BIT20 := FALSE;
   STATUS[194].EXT.AlarmSuppressed := FALSE;
   STATUS[194].EXT.AlarmPresent := FALSE;
   STATUS[194].EXT.AlarmFailUnAck := FALSE;
   STATUS[194].Status := 0;
   STATUS[194].TimeStamp := 16#0000;
   STATUS[195].EXT.AlarmWarnUnAck := FALSE;
   STATUS[195].EXT.AckRequired := FALSE;
   STATUS[195].EXT.Maintanence := FALSE;
   STATUS[195].EXT.Operation := FALSE;
   STATUS[195].EXT.Forced := FALSE;
   STATUS[195].EXT.BIT29 := FALSE;
   STATUS[195].EXT.BIT30 := FALSE;
   STATUS[195].EXT.BIT31 := FALSE;
   STATUS[195].EXT.ModeBit1 := FALSE;
   STATUS[195].EXT.ModeBit2 := FALSE;
   STATUS[195].EXT.ModeBit3 := FALSE;
   STATUS[195].EXT.BIT19 := FALSE;
   STATUS[195].EXT.BIT20 := FALSE;
   STATUS[195].EXT.AlarmSuppressed := FALSE;
   STATUS[195].EXT.AlarmPresent := FALSE;
   STATUS[195].EXT.AlarmFailUnAck := FALSE;
   STATUS[195].Status := 0;
   STATUS[195].TimeStamp := 16#0000;
   STATUS[196].EXT.AlarmWarnUnAck := FALSE;
   STATUS[196].EXT.AckRequired := FALSE;
   STATUS[196].EXT.Maintanence := FALSE;
   STATUS[196].EXT.Operation := FALSE;
   STATUS[196].EXT.Forced := FALSE;
   STATUS[196].EXT.BIT29 := FALSE;
   STATUS[196].EXT.BIT30 := FALSE;
   STATUS[196].EXT.BIT31 := FALSE;
   STATUS[196].EXT.ModeBit1 := FALSE;
   STATUS[196].EXT.ModeBit2 := FALSE;
   STATUS[196].EXT.ModeBit3 := FALSE;
   STATUS[196].EXT.BIT19 := FALSE;
   STATUS[196].EXT.BIT20 := FALSE;
   STATUS[196].EXT.AlarmSuppressed := FALSE;
   STATUS[196].EXT.AlarmPresent := FALSE;
   STATUS[196].EXT.AlarmFailUnAck := FALSE;
   STATUS[196].Status := 0;
   STATUS[196].TimeStamp := 16#0000;
   STATUS[197].EXT.AlarmWarnUnAck := FALSE;
   STATUS[197].EXT.AckRequired := FALSE;
   STATUS[197].EXT.Maintanence := FALSE;
   STATUS[197].EXT.Operation := FALSE;
   STATUS[197].EXT.Forced := FALSE;
   STATUS[197].EXT.BIT29 := FALSE;
   STATUS[197].EXT.BIT30 := FALSE;
   STATUS[197].EXT.BIT31 := FALSE;
   STATUS[197].EXT.ModeBit1 := FALSE;
   STATUS[197].EXT.ModeBit2 := FALSE;
   STATUS[197].EXT.ModeBit3 := FALSE;
   STATUS[197].EXT.BIT19 := FALSE;
   STATUS[197].EXT.BIT20 := FALSE;
   STATUS[197].EXT.AlarmSuppressed := FALSE;
   STATUS[197].EXT.AlarmPresent := FALSE;
   STATUS[197].EXT.AlarmFailUnAck := FALSE;
   STATUS[197].Status := 0;
   STATUS[197].TimeStamp := 16#0000;
   STATUS[198].EXT.AlarmWarnUnAck := FALSE;
   STATUS[198].EXT.AckRequired := FALSE;
   STATUS[198].EXT.Maintanence := FALSE;
   STATUS[198].EXT.Operation := FALSE;
   STATUS[198].EXT.Forced := FALSE;
   STATUS[198].EXT.BIT29 := FALSE;
   STATUS[198].EXT.BIT30 := FALSE;
   STATUS[198].EXT.BIT31 := FALSE;
   STATUS[198].EXT.ModeBit1 := FALSE;
   STATUS[198].EXT.ModeBit2 := FALSE;
   STATUS[198].EXT.ModeBit3 := FALSE;
   STATUS[198].EXT.BIT19 := FALSE;
   STATUS[198].EXT.BIT20 := FALSE;
   STATUS[198].EXT.AlarmSuppressed := FALSE;
   STATUS[198].EXT.AlarmPresent := FALSE;
   STATUS[198].EXT.AlarmFailUnAck := FALSE;
   STATUS[198].Status := 0;
   STATUS[198].TimeStamp := 16#0000;
   STATUS[199].EXT.AlarmWarnUnAck := FALSE;
   STATUS[199].EXT.AckRequired := FALSE;
   STATUS[199].EXT.Maintanence := FALSE;
   STATUS[199].EXT.Operation := FALSE;
   STATUS[199].EXT.Forced := FALSE;
   STATUS[199].EXT.BIT29 := FALSE;
   STATUS[199].EXT.BIT30 := FALSE;
   STATUS[199].EXT.BIT31 := FALSE;
   STATUS[199].EXT.ModeBit1 := FALSE;
   STATUS[199].EXT.ModeBit2 := FALSE;
   STATUS[199].EXT.ModeBit3 := FALSE;
   STATUS[199].EXT.BIT19 := FALSE;
   STATUS[199].EXT.BIT20 := FALSE;
   STATUS[199].EXT.AlarmSuppressed := FALSE;
   STATUS[199].EXT.AlarmPresent := FALSE;
   STATUS[199].EXT.AlarmFailUnAck := FALSE;
   STATUS[199].Status := 0;
   STATUS[199].TimeStamp := 16#0000;
   STATUS[200].EXT.AlarmWarnUnAck := FALSE;
   STATUS[200].EXT.AckRequired := TRUE;
   STATUS[200].EXT.Maintanence := FALSE;
   STATUS[200].EXT.Operation := TRUE;
   STATUS[200].EXT.Forced := FALSE;
   STATUS[200].EXT.BIT29 := FALSE;
   STATUS[200].EXT.BIT30 := FALSE;
   STATUS[200].EXT.BIT31 := FALSE;
   STATUS[200].EXT.ModeBit1 := FALSE;
   STATUS[200].EXT.ModeBit2 := FALSE;
   STATUS[200].EXT.ModeBit3 := FALSE;
   STATUS[200].EXT.BIT19 := FALSE;
   STATUS[200].EXT.BIT20 := FALSE;
   STATUS[200].EXT.AlarmSuppressed := FALSE;
   STATUS[200].EXT.AlarmPresent := FALSE;
   STATUS[200].EXT.AlarmFailUnAck := TRUE;
   STATUS[200].Status := 10;
   STATUS[200].TimeStamp := 16#A4CC;
   STATUS[201].EXT.AlarmWarnUnAck := FALSE;
   STATUS[201].EXT.AckRequired := FALSE;
   STATUS[201].EXT.Maintanence := FALSE;
   STATUS[201].EXT.Operation := FALSE;
   STATUS[201].EXT.Forced := FALSE;
   STATUS[201].EXT.BIT29 := FALSE;
   STATUS[201].EXT.BIT30 := FALSE;
   STATUS[201].EXT.BIT31 := FALSE;
   STATUS[201].EXT.ModeBit1 := FALSE;
   STATUS[201].EXT.ModeBit2 := FALSE;
   STATUS[201].EXT.ModeBit3 := FALSE;
   STATUS[201].EXT.BIT19 := FALSE;
   STATUS[201].EXT.BIT20 := FALSE;
   STATUS[201].EXT.AlarmSuppressed := FALSE;
   STATUS[201].EXT.AlarmPresent := FALSE;
   STATUS[201].EXT.AlarmFailUnAck := FALSE;
   STATUS[201].Status := 0;
   STATUS[201].TimeStamp := 16#0000;
   STATUS[202].EXT.AlarmWarnUnAck := FALSE;
   STATUS[202].EXT.AckRequired := FALSE;
   STATUS[202].EXT.Maintanence := FALSE;
   STATUS[202].EXT.Operation := FALSE;
   STATUS[202].EXT.Forced := FALSE;
   STATUS[202].EXT.BIT29 := FALSE;
   STATUS[202].EXT.BIT30 := FALSE;
   STATUS[202].EXT.BIT31 := FALSE;
   STATUS[202].EXT.ModeBit1 := FALSE;
   STATUS[202].EXT.ModeBit2 := FALSE;
   STATUS[202].EXT.ModeBit3 := FALSE;
   STATUS[202].EXT.BIT19 := FALSE;
   STATUS[202].EXT.BIT20 := FALSE;
   STATUS[202].EXT.AlarmSuppressed := FALSE;
   STATUS[202].EXT.AlarmPresent := FALSE;
   STATUS[202].EXT.AlarmFailUnAck := FALSE;
   STATUS[202].Status := 0;
   STATUS[202].TimeStamp := 16#0000;
   STATUS[203].EXT.AlarmWarnUnAck := FALSE;
   STATUS[203].EXT.AckRequired := FALSE;
   STATUS[203].EXT.Maintanence := FALSE;
   STATUS[203].EXT.Operation := FALSE;
   STATUS[203].EXT.Forced := FALSE;
   STATUS[203].EXT.BIT29 := FALSE;
   STATUS[203].EXT.BIT30 := FALSE;
   STATUS[203].EXT.BIT31 := FALSE;
   STATUS[203].EXT.ModeBit1 := FALSE;
   STATUS[203].EXT.ModeBit2 := FALSE;
   STATUS[203].EXT.ModeBit3 := FALSE;
   STATUS[203].EXT.BIT19 := FALSE;
   STATUS[203].EXT.BIT20 := FALSE;
   STATUS[203].EXT.AlarmSuppressed := FALSE;
   STATUS[203].EXT.AlarmPresent := FALSE;
   STATUS[203].EXT.AlarmFailUnAck := FALSE;
   STATUS[203].Status := 0;
   STATUS[203].TimeStamp := 16#0000;
   STATUS[204].EXT.AlarmWarnUnAck := FALSE;
   STATUS[204].EXT.AckRequired := FALSE;
   STATUS[204].EXT.Maintanence := FALSE;
   STATUS[204].EXT.Operation := FALSE;
   STATUS[204].EXT.Forced := FALSE;
   STATUS[204].EXT.BIT29 := FALSE;
   STATUS[204].EXT.BIT30 := FALSE;
   STATUS[204].EXT.BIT31 := FALSE;
   STATUS[204].EXT.ModeBit1 := FALSE;
   STATUS[204].EXT.ModeBit2 := FALSE;
   STATUS[204].EXT.ModeBit3 := FALSE;
   STATUS[204].EXT.BIT19 := FALSE;
   STATUS[204].EXT.BIT20 := FALSE;
   STATUS[204].EXT.AlarmSuppressed := FALSE;
   STATUS[204].EXT.AlarmPresent := FALSE;
   STATUS[204].EXT.AlarmFailUnAck := FALSE;
   STATUS[204].Status := 0;
   STATUS[204].TimeStamp := 16#0000;
   STATUS[205].EXT.AlarmWarnUnAck := FALSE;
   STATUS[205].EXT.AckRequired := FALSE;
   STATUS[205].EXT.Maintanence := FALSE;
   STATUS[205].EXT.Operation := FALSE;
   STATUS[205].EXT.Forced := FALSE;
   STATUS[205].EXT.BIT29 := FALSE;
   STATUS[205].EXT.BIT30 := FALSE;
   STATUS[205].EXT.BIT31 := FALSE;
   STATUS[205].EXT.ModeBit1 := FALSE;
   STATUS[205].EXT.ModeBit2 := FALSE;
   STATUS[205].EXT.ModeBit3 := FALSE;
   STATUS[205].EXT.BIT19 := FALSE;
   STATUS[205].EXT.BIT20 := FALSE;
   STATUS[205].EXT.AlarmSuppressed := FALSE;
   STATUS[205].EXT.AlarmPresent := FALSE;
   STATUS[205].EXT.AlarmFailUnAck := FALSE;
   STATUS[205].Status := 0;
   STATUS[205].TimeStamp := 16#0000;
   STATUS[206].EXT.AlarmWarnUnAck := FALSE;
   STATUS[206].EXT.AckRequired := FALSE;
   STATUS[206].EXT.Maintanence := FALSE;
   STATUS[206].EXT.Operation := FALSE;
   STATUS[206].EXT.Forced := FALSE;
   STATUS[206].EXT.BIT29 := FALSE;
   STATUS[206].EXT.BIT30 := FALSE;
   STATUS[206].EXT.BIT31 := FALSE;
   STATUS[206].EXT.ModeBit1 := FALSE;
   STATUS[206].EXT.ModeBit2 := FALSE;
   STATUS[206].EXT.ModeBit3 := FALSE;
   STATUS[206].EXT.BIT19 := FALSE;
   STATUS[206].EXT.BIT20 := FALSE;
   STATUS[206].EXT.AlarmSuppressed := FALSE;
   STATUS[206].EXT.AlarmPresent := FALSE;
   STATUS[206].EXT.AlarmFailUnAck := FALSE;
   STATUS[206].Status := 0;
   STATUS[206].TimeStamp := 16#0000;
   STATUS[207].EXT.AlarmWarnUnAck := FALSE;
   STATUS[207].EXT.AckRequired := FALSE;
   STATUS[207].EXT.Maintanence := FALSE;
   STATUS[207].EXT.Operation := FALSE;
   STATUS[207].EXT.Forced := FALSE;
   STATUS[207].EXT.BIT29 := FALSE;
   STATUS[207].EXT.BIT30 := FALSE;
   STATUS[207].EXT.BIT31 := FALSE;
   STATUS[207].EXT.ModeBit1 := FALSE;
   STATUS[207].EXT.ModeBit2 := FALSE;
   STATUS[207].EXT.ModeBit3 := FALSE;
   STATUS[207].EXT.BIT19 := FALSE;
   STATUS[207].EXT.BIT20 := FALSE;
   STATUS[207].EXT.AlarmSuppressed := FALSE;
   STATUS[207].EXT.AlarmPresent := FALSE;
   STATUS[207].EXT.AlarmFailUnAck := FALSE;
   STATUS[207].Status := 0;
   STATUS[207].TimeStamp := 16#0000;
   STATUS[208].EXT.AlarmWarnUnAck := FALSE;
   STATUS[208].EXT.AckRequired := FALSE;
   STATUS[208].EXT.Maintanence := FALSE;
   STATUS[208].EXT.Operation := FALSE;
   STATUS[208].EXT.Forced := FALSE;
   STATUS[208].EXT.BIT29 := FALSE;
   STATUS[208].EXT.BIT30 := FALSE;
   STATUS[208].EXT.BIT31 := FALSE;
   STATUS[208].EXT.ModeBit1 := FALSE;
   STATUS[208].EXT.ModeBit2 := FALSE;
   STATUS[208].EXT.ModeBit3 := FALSE;
   STATUS[208].EXT.BIT19 := FALSE;
   STATUS[208].EXT.BIT20 := FALSE;
   STATUS[208].EXT.AlarmSuppressed := FALSE;
   STATUS[208].EXT.AlarmPresent := FALSE;
   STATUS[208].EXT.AlarmFailUnAck := FALSE;
   STATUS[208].Status := 0;
   STATUS[208].TimeStamp := 16#0000;
   STATUS[209].EXT.AlarmWarnUnAck := FALSE;
   STATUS[209].EXT.AckRequired := FALSE;
   STATUS[209].EXT.Maintanence := FALSE;
   STATUS[209].EXT.Operation := FALSE;
   STATUS[209].EXT.Forced := FALSE;
   STATUS[209].EXT.BIT29 := FALSE;
   STATUS[209].EXT.BIT30 := FALSE;
   STATUS[209].EXT.BIT31 := FALSE;
   STATUS[209].EXT.ModeBit1 := FALSE;
   STATUS[209].EXT.ModeBit2 := FALSE;
   STATUS[209].EXT.ModeBit3 := FALSE;
   STATUS[209].EXT.BIT19 := FALSE;
   STATUS[209].EXT.BIT20 := FALSE;
   STATUS[209].EXT.AlarmSuppressed := FALSE;
   STATUS[209].EXT.AlarmPresent := FALSE;
   STATUS[209].EXT.AlarmFailUnAck := FALSE;
   STATUS[209].Status := 0;
   STATUS[209].TimeStamp := 16#0000;
   STATUS[210].EXT.AlarmWarnUnAck := FALSE;
   STATUS[210].EXT.AckRequired := FALSE;
   STATUS[210].EXT.Maintanence := FALSE;
   STATUS[210].EXT.Operation := FALSE;
   STATUS[210].EXT.Forced := FALSE;
   STATUS[210].EXT.BIT29 := FALSE;
   STATUS[210].EXT.BIT30 := FALSE;
   STATUS[210].EXT.BIT31 := FALSE;
   STATUS[210].EXT.ModeBit1 := FALSE;
   STATUS[210].EXT.ModeBit2 := FALSE;
   STATUS[210].EXT.ModeBit3 := FALSE;
   STATUS[210].EXT.BIT19 := FALSE;
   STATUS[210].EXT.BIT20 := FALSE;
   STATUS[210].EXT.AlarmSuppressed := FALSE;
   STATUS[210].EXT.AlarmPresent := FALSE;
   STATUS[210].EXT.AlarmFailUnAck := FALSE;
   STATUS[210].Status := 0;
   STATUS[210].TimeStamp := 16#0000;
   STATUS[211].EXT.AlarmWarnUnAck := FALSE;
   STATUS[211].EXT.AckRequired := FALSE;
   STATUS[211].EXT.Maintanence := FALSE;
   STATUS[211].EXT.Operation := FALSE;
   STATUS[211].EXT.Forced := FALSE;
   STATUS[211].EXT.BIT29 := FALSE;
   STATUS[211].EXT.BIT30 := FALSE;
   STATUS[211].EXT.BIT31 := FALSE;
   STATUS[211].EXT.ModeBit1 := FALSE;
   STATUS[211].EXT.ModeBit2 := FALSE;
   STATUS[211].EXT.ModeBit3 := FALSE;
   STATUS[211].EXT.BIT19 := FALSE;
   STATUS[211].EXT.BIT20 := FALSE;
   STATUS[211].EXT.AlarmSuppressed := FALSE;
   STATUS[211].EXT.AlarmPresent := FALSE;
   STATUS[211].EXT.AlarmFailUnAck := FALSE;
   STATUS[211].Status := 0;
   STATUS[211].TimeStamp := 16#0000;
   STATUS[212].EXT.AlarmWarnUnAck := FALSE;
   STATUS[212].EXT.AckRequired := FALSE;
   STATUS[212].EXT.Maintanence := FALSE;
   STATUS[212].EXT.Operation := FALSE;
   STATUS[212].EXT.Forced := FALSE;
   STATUS[212].EXT.BIT29 := FALSE;
   STATUS[212].EXT.BIT30 := FALSE;
   STATUS[212].EXT.BIT31 := FALSE;
   STATUS[212].EXT.ModeBit1 := FALSE;
   STATUS[212].EXT.ModeBit2 := FALSE;
   STATUS[212].EXT.ModeBit3 := FALSE;
   STATUS[212].EXT.BIT19 := FALSE;
   STATUS[212].EXT.BIT20 := FALSE;
   STATUS[212].EXT.AlarmSuppressed := FALSE;
   STATUS[212].EXT.AlarmPresent := FALSE;
   STATUS[212].EXT.AlarmFailUnAck := FALSE;
   STATUS[212].Status := 0;
   STATUS[212].TimeStamp := 16#0000;
   STATUS[213].EXT.AlarmWarnUnAck := FALSE;
   STATUS[213].EXT.AckRequired := FALSE;
   STATUS[213].EXT.Maintanence := FALSE;
   STATUS[213].EXT.Operation := FALSE;
   STATUS[213].EXT.Forced := FALSE;
   STATUS[213].EXT.BIT29 := FALSE;
   STATUS[213].EXT.BIT30 := FALSE;
   STATUS[213].EXT.BIT31 := FALSE;
   STATUS[213].EXT.ModeBit1 := FALSE;
   STATUS[213].EXT.ModeBit2 := FALSE;
   STATUS[213].EXT.ModeBit3 := FALSE;
   STATUS[213].EXT.BIT19 := FALSE;
   STATUS[213].EXT.BIT20 := FALSE;
   STATUS[213].EXT.AlarmSuppressed := FALSE;
   STATUS[213].EXT.AlarmPresent := FALSE;
   STATUS[213].EXT.AlarmFailUnAck := FALSE;
   STATUS[213].Status := 0;
   STATUS[213].TimeStamp := 16#0000;
   STATUS[214].EXT.AlarmWarnUnAck := FALSE;
   STATUS[214].EXT.AckRequired := FALSE;
   STATUS[214].EXT.Maintanence := FALSE;
   STATUS[214].EXT.Operation := FALSE;
   STATUS[214].EXT.Forced := FALSE;
   STATUS[214].EXT.BIT29 := FALSE;
   STATUS[214].EXT.BIT30 := FALSE;
   STATUS[214].EXT.BIT31 := FALSE;
   STATUS[214].EXT.ModeBit1 := FALSE;
   STATUS[214].EXT.ModeBit2 := FALSE;
   STATUS[214].EXT.ModeBit3 := FALSE;
   STATUS[214].EXT.BIT19 := FALSE;
   STATUS[214].EXT.BIT20 := FALSE;
   STATUS[214].EXT.AlarmSuppressed := FALSE;
   STATUS[214].EXT.AlarmPresent := FALSE;
   STATUS[214].EXT.AlarmFailUnAck := FALSE;
   STATUS[214].Status := 0;
   STATUS[214].TimeStamp := 16#0000;
   STATUS[215].EXT.AlarmWarnUnAck := FALSE;
   STATUS[215].EXT.AckRequired := FALSE;
   STATUS[215].EXT.Maintanence := FALSE;
   STATUS[215].EXT.Operation := FALSE;
   STATUS[215].EXT.Forced := FALSE;
   STATUS[215].EXT.BIT29 := FALSE;
   STATUS[215].EXT.BIT30 := FALSE;
   STATUS[215].EXT.BIT31 := FALSE;
   STATUS[215].EXT.ModeBit1 := FALSE;
   STATUS[215].EXT.ModeBit2 := FALSE;
   STATUS[215].EXT.ModeBit3 := FALSE;
   STATUS[215].EXT.BIT19 := FALSE;
   STATUS[215].EXT.BIT20 := FALSE;
   STATUS[215].EXT.AlarmSuppressed := FALSE;
   STATUS[215].EXT.AlarmPresent := FALSE;
   STATUS[215].EXT.AlarmFailUnAck := FALSE;
   STATUS[215].Status := 0;
   STATUS[215].TimeStamp := 16#0000;
   STATUS[216].EXT.AlarmWarnUnAck := FALSE;
   STATUS[216].EXT.AckRequired := FALSE;
   STATUS[216].EXT.Maintanence := FALSE;
   STATUS[216].EXT.Operation := FALSE;
   STATUS[216].EXT.Forced := FALSE;
   STATUS[216].EXT.BIT29 := FALSE;
   STATUS[216].EXT.BIT30 := FALSE;
   STATUS[216].EXT.BIT31 := FALSE;
   STATUS[216].EXT.ModeBit1 := FALSE;
   STATUS[216].EXT.ModeBit2 := FALSE;
   STATUS[216].EXT.ModeBit3 := FALSE;
   STATUS[216].EXT.BIT19 := FALSE;
   STATUS[216].EXT.BIT20 := FALSE;
   STATUS[216].EXT.AlarmSuppressed := FALSE;
   STATUS[216].EXT.AlarmPresent := FALSE;
   STATUS[216].EXT.AlarmFailUnAck := FALSE;
   STATUS[216].Status := 0;
   STATUS[216].TimeStamp := 16#0000;
   STATUS[217].EXT.AlarmWarnUnAck := FALSE;
   STATUS[217].EXT.AckRequired := FALSE;
   STATUS[217].EXT.Maintanence := FALSE;
   STATUS[217].EXT.Operation := FALSE;
   STATUS[217].EXT.Forced := FALSE;
   STATUS[217].EXT.BIT29 := FALSE;
   STATUS[217].EXT.BIT30 := FALSE;
   STATUS[217].EXT.BIT31 := FALSE;
   STATUS[217].EXT.ModeBit1 := FALSE;
   STATUS[217].EXT.ModeBit2 := FALSE;
   STATUS[217].EXT.ModeBit3 := FALSE;
   STATUS[217].EXT.BIT19 := FALSE;
   STATUS[217].EXT.BIT20 := FALSE;
   STATUS[217].EXT.AlarmSuppressed := FALSE;
   STATUS[217].EXT.AlarmPresent := FALSE;
   STATUS[217].EXT.AlarmFailUnAck := FALSE;
   STATUS[217].Status := 0;
   STATUS[217].TimeStamp := 16#0000;
   STATUS[218].EXT.AlarmWarnUnAck := FALSE;
   STATUS[218].EXT.AckRequired := FALSE;
   STATUS[218].EXT.Maintanence := FALSE;
   STATUS[218].EXT.Operation := FALSE;
   STATUS[218].EXT.Forced := FALSE;
   STATUS[218].EXT.BIT29 := FALSE;
   STATUS[218].EXT.BIT30 := FALSE;
   STATUS[218].EXT.BIT31 := FALSE;
   STATUS[218].EXT.ModeBit1 := FALSE;
   STATUS[218].EXT.ModeBit2 := FALSE;
   STATUS[218].EXT.ModeBit3 := FALSE;
   STATUS[218].EXT.BIT19 := FALSE;
   STATUS[218].EXT.BIT20 := FALSE;
   STATUS[218].EXT.AlarmSuppressed := FALSE;
   STATUS[218].EXT.AlarmPresent := FALSE;
   STATUS[218].EXT.AlarmFailUnAck := FALSE;
   STATUS[218].Status := 0;
   STATUS[218].TimeStamp := 16#0000;
   STATUS[219].EXT.AlarmWarnUnAck := FALSE;
   STATUS[219].EXT.AckRequired := FALSE;
   STATUS[219].EXT.Maintanence := FALSE;
   STATUS[219].EXT.Operation := FALSE;
   STATUS[219].EXT.Forced := FALSE;
   STATUS[219].EXT.BIT29 := FALSE;
   STATUS[219].EXT.BIT30 := FALSE;
   STATUS[219].EXT.BIT31 := FALSE;
   STATUS[219].EXT.ModeBit1 := FALSE;
   STATUS[219].EXT.ModeBit2 := FALSE;
   STATUS[219].EXT.ModeBit3 := FALSE;
   STATUS[219].EXT.BIT19 := FALSE;
   STATUS[219].EXT.BIT20 := FALSE;
   STATUS[219].EXT.AlarmSuppressed := FALSE;
   STATUS[219].EXT.AlarmPresent := FALSE;
   STATUS[219].EXT.AlarmFailUnAck := FALSE;
   STATUS[219].Status := 0;
   STATUS[219].TimeStamp := 16#0000;
   STATUS[220].EXT.AlarmWarnUnAck := FALSE;
   STATUS[220].EXT.AckRequired := FALSE;
   STATUS[220].EXT.Maintanence := FALSE;
   STATUS[220].EXT.Operation := FALSE;
   STATUS[220].EXT.Forced := FALSE;
   STATUS[220].EXT.BIT29 := FALSE;
   STATUS[220].EXT.BIT30 := FALSE;
   STATUS[220].EXT.BIT31 := FALSE;
   STATUS[220].EXT.ModeBit1 := FALSE;
   STATUS[220].EXT.ModeBit2 := FALSE;
   STATUS[220].EXT.ModeBit3 := FALSE;
   STATUS[220].EXT.BIT19 := FALSE;
   STATUS[220].EXT.BIT20 := FALSE;
   STATUS[220].EXT.AlarmSuppressed := FALSE;
   STATUS[220].EXT.AlarmPresent := FALSE;
   STATUS[220].EXT.AlarmFailUnAck := FALSE;
   STATUS[220].Status := 0;
   STATUS[220].TimeStamp := 16#0000;
   STATUS[221].EXT.AlarmWarnUnAck := FALSE;
   STATUS[221].EXT.AckRequired := FALSE;
   STATUS[221].EXT.Maintanence := FALSE;
   STATUS[221].EXT.Operation := FALSE;
   STATUS[221].EXT.Forced := FALSE;
   STATUS[221].EXT.BIT29 := FALSE;
   STATUS[221].EXT.BIT30 := FALSE;
   STATUS[221].EXT.BIT31 := FALSE;
   STATUS[221].EXT.ModeBit1 := FALSE;
   STATUS[221].EXT.ModeBit2 := FALSE;
   STATUS[221].EXT.ModeBit3 := FALSE;
   STATUS[221].EXT.BIT19 := FALSE;
   STATUS[221].EXT.BIT20 := FALSE;
   STATUS[221].EXT.AlarmSuppressed := FALSE;
   STATUS[221].EXT.AlarmPresent := FALSE;
   STATUS[221].EXT.AlarmFailUnAck := FALSE;
   STATUS[221].Status := 0;
   STATUS[221].TimeStamp := 16#0000;
   STATUS[222].EXT.AlarmWarnUnAck := FALSE;
   STATUS[222].EXT.AckRequired := FALSE;
   STATUS[222].EXT.Maintanence := FALSE;
   STATUS[222].EXT.Operation := FALSE;
   STATUS[222].EXT.Forced := FALSE;
   STATUS[222].EXT.BIT29 := FALSE;
   STATUS[222].EXT.BIT30 := FALSE;
   STATUS[222].EXT.BIT31 := FALSE;
   STATUS[222].EXT.ModeBit1 := FALSE;
   STATUS[222].EXT.ModeBit2 := FALSE;
   STATUS[222].EXT.ModeBit3 := FALSE;
   STATUS[222].EXT.BIT19 := FALSE;
   STATUS[222].EXT.BIT20 := FALSE;
   STATUS[222].EXT.AlarmSuppressed := FALSE;
   STATUS[222].EXT.AlarmPresent := FALSE;
   STATUS[222].EXT.AlarmFailUnAck := FALSE;
   STATUS[222].Status := 0;
   STATUS[222].TimeStamp := 16#0000;
   STATUS[223].EXT.AlarmWarnUnAck := FALSE;
   STATUS[223].EXT.AckRequired := FALSE;
   STATUS[223].EXT.Maintanence := FALSE;
   STATUS[223].EXT.Operation := FALSE;
   STATUS[223].EXT.Forced := FALSE;
   STATUS[223].EXT.BIT29 := FALSE;
   STATUS[223].EXT.BIT30 := FALSE;
   STATUS[223].EXT.BIT31 := FALSE;
   STATUS[223].EXT.ModeBit1 := FALSE;
   STATUS[223].EXT.ModeBit2 := FALSE;
   STATUS[223].EXT.ModeBit3 := FALSE;
   STATUS[223].EXT.BIT19 := FALSE;
   STATUS[223].EXT.BIT20 := FALSE;
   STATUS[223].EXT.AlarmSuppressed := FALSE;
   STATUS[223].EXT.AlarmPresent := FALSE;
   STATUS[223].EXT.AlarmFailUnAck := FALSE;
   STATUS[223].Status := 0;
   STATUS[223].TimeStamp := 16#0000;
   STATUS[224].EXT.AlarmWarnUnAck := FALSE;
   STATUS[224].EXT.AckRequired := FALSE;
   STATUS[224].EXT.Maintanence := FALSE;
   STATUS[224].EXT.Operation := FALSE;
   STATUS[224].EXT.Forced := FALSE;
   STATUS[224].EXT.BIT29 := FALSE;
   STATUS[224].EXT.BIT30 := FALSE;
   STATUS[224].EXT.BIT31 := FALSE;
   STATUS[224].EXT.ModeBit1 := FALSE;
   STATUS[224].EXT.ModeBit2 := FALSE;
   STATUS[224].EXT.ModeBit3 := FALSE;
   STATUS[224].EXT.BIT19 := FALSE;
   STATUS[224].EXT.BIT20 := FALSE;
   STATUS[224].EXT.AlarmSuppressed := FALSE;
   STATUS[224].EXT.AlarmPresent := FALSE;
   STATUS[224].EXT.AlarmFailUnAck := FALSE;
   STATUS[224].Status := 0;
   STATUS[224].TimeStamp := 16#0000;
   STATUS[225].EXT.AlarmWarnUnAck := FALSE;
   STATUS[225].EXT.AckRequired := FALSE;
   STATUS[225].EXT.Maintanence := FALSE;
   STATUS[225].EXT.Operation := FALSE;
   STATUS[225].EXT.Forced := FALSE;
   STATUS[225].EXT.BIT29 := FALSE;
   STATUS[225].EXT.BIT30 := FALSE;
   STATUS[225].EXT.BIT31 := FALSE;
   STATUS[225].EXT.ModeBit1 := FALSE;
   STATUS[225].EXT.ModeBit2 := FALSE;
   STATUS[225].EXT.ModeBit3 := FALSE;
   STATUS[225].EXT.BIT19 := FALSE;
   STATUS[225].EXT.BIT20 := FALSE;
   STATUS[225].EXT.AlarmSuppressed := FALSE;
   STATUS[225].EXT.AlarmPresent := FALSE;
   STATUS[225].EXT.AlarmFailUnAck := FALSE;
   STATUS[225].Status := 0;
   STATUS[225].TimeStamp := 16#0000;
   STATUS[226].EXT.AlarmWarnUnAck := FALSE;
   STATUS[226].EXT.AckRequired := FALSE;
   STATUS[226].EXT.Maintanence := FALSE;
   STATUS[226].EXT.Operation := FALSE;
   STATUS[226].EXT.Forced := FALSE;
   STATUS[226].EXT.BIT29 := FALSE;
   STATUS[226].EXT.BIT30 := FALSE;
   STATUS[226].EXT.BIT31 := FALSE;
   STATUS[226].EXT.ModeBit1 := FALSE;
   STATUS[226].EXT.ModeBit2 := FALSE;
   STATUS[226].EXT.ModeBit3 := FALSE;
   STATUS[226].EXT.BIT19 := FALSE;
   STATUS[226].EXT.BIT20 := FALSE;
   STATUS[226].EXT.AlarmSuppressed := FALSE;
   STATUS[226].EXT.AlarmPresent := FALSE;
   STATUS[226].EXT.AlarmFailUnAck := FALSE;
   STATUS[226].Status := 0;
   STATUS[226].TimeStamp := 16#0000;
   STATUS[227].EXT.AlarmWarnUnAck := FALSE;
   STATUS[227].EXT.AckRequired := FALSE;
   STATUS[227].EXT.Maintanence := FALSE;
   STATUS[227].EXT.Operation := FALSE;
   STATUS[227].EXT.Forced := FALSE;
   STATUS[227].EXT.BIT29 := FALSE;
   STATUS[227].EXT.BIT30 := FALSE;
   STATUS[227].EXT.BIT31 := FALSE;
   STATUS[227].EXT.ModeBit1 := FALSE;
   STATUS[227].EXT.ModeBit2 := FALSE;
   STATUS[227].EXT.ModeBit3 := FALSE;
   STATUS[227].EXT.BIT19 := FALSE;
   STATUS[227].EXT.BIT20 := FALSE;
   STATUS[227].EXT.AlarmSuppressed := FALSE;
   STATUS[227].EXT.AlarmPresent := FALSE;
   STATUS[227].EXT.AlarmFailUnAck := FALSE;
   STATUS[227].Status := 0;
   STATUS[227].TimeStamp := 16#0000;
   STATUS[228].EXT.AlarmWarnUnAck := FALSE;
   STATUS[228].EXT.AckRequired := FALSE;
   STATUS[228].EXT.Maintanence := FALSE;
   STATUS[228].EXT.Operation := FALSE;
   STATUS[228].EXT.Forced := FALSE;
   STATUS[228].EXT.BIT29 := FALSE;
   STATUS[228].EXT.BIT30 := FALSE;
   STATUS[228].EXT.BIT31 := FALSE;
   STATUS[228].EXT.ModeBit1 := FALSE;
   STATUS[228].EXT.ModeBit2 := FALSE;
   STATUS[228].EXT.ModeBit3 := FALSE;
   STATUS[228].EXT.BIT19 := FALSE;
   STATUS[228].EXT.BIT20 := FALSE;
   STATUS[228].EXT.AlarmSuppressed := FALSE;
   STATUS[228].EXT.AlarmPresent := FALSE;
   STATUS[228].EXT.AlarmFailUnAck := FALSE;
   STATUS[228].Status := 0;
   STATUS[228].TimeStamp := 16#0000;
   STATUS[229].EXT.AlarmWarnUnAck := FALSE;
   STATUS[229].EXT.AckRequired := FALSE;
   STATUS[229].EXT.Maintanence := FALSE;
   STATUS[229].EXT.Operation := FALSE;
   STATUS[229].EXT.Forced := FALSE;
   STATUS[229].EXT.BIT29 := FALSE;
   STATUS[229].EXT.BIT30 := FALSE;
   STATUS[229].EXT.BIT31 := FALSE;
   STATUS[229].EXT.ModeBit1 := FALSE;
   STATUS[229].EXT.ModeBit2 := FALSE;
   STATUS[229].EXT.ModeBit3 := FALSE;
   STATUS[229].EXT.BIT19 := FALSE;
   STATUS[229].EXT.BIT20 := FALSE;
   STATUS[229].EXT.AlarmSuppressed := FALSE;
   STATUS[229].EXT.AlarmPresent := FALSE;
   STATUS[229].EXT.AlarmFailUnAck := FALSE;
   STATUS[229].Status := 0;
   STATUS[229].TimeStamp := 16#0000;
   STATUS[230].EXT.AlarmWarnUnAck := FALSE;
   STATUS[230].EXT.AckRequired := FALSE;
   STATUS[230].EXT.Maintanence := FALSE;
   STATUS[230].EXT.Operation := FALSE;
   STATUS[230].EXT.Forced := FALSE;
   STATUS[230].EXT.BIT29 := FALSE;
